TEXTLIST S3_Alarms
  0 = 'Station 3 Clamp A1 Failed to Advance... Check Q1.0...' | German: 'S3 0 Row 1 Failed To Advance.. Check Qxxx.x German' | French: 'S3 0 Row 1 Failed To Advance.. Check Qxxx.x French' | 汉语: '汉语'
  1 = 'Station 3 Clamp A1 Failed to Return... Check Q1.1...' | German: 'S3 1 Row 1 Failed To Return.. Check Qxxx.x German' | French: 'S3 1 Row 1 Failed To Return.. Check Qxxx.x French' | 汉语: '汉语'
  2 = 'Station 3 Clamp A1 Lost Advanced... Check I1.0...' | German: 'S3 2 Row 1 Lost Advance Position... Check Ixxx.x German' | French: 'S3 2 Row 1 Lost Advance Position... Check Ixxx.x French' | 汉语: '汉语'
  3 = 'Station 3 Clamp A1 Lost Returned... Check I1.1...' | German: 'S3 3 Row 1 Lost Return Position... Check Ixxx.x German' | French: 'S3 3 Row 1 Lost Return Position... Check Ixxx.x French' | 汉语: '汉语'
  4 = 'Station 3 Clamp A1 Switch Fault... Check I1.0, I1.1...' | German: 'S3 4 Row 1 Switch Fault... Check Ixxx.x / Ixxx.x German' | French: 'S3 4 Row 1 Switch Fault... Check Ixxx.x / Ixxx.x French' | 汉语: '汉语'
  5 = 'Spare' | German: 'S3 5 Row 1 Spare Message German' | French: 'S3 5 Row 1 Spare Message French'
  6 = 'Spare' | German: 'S3 6 Row 1 Spare Message German' | French: 'S3 6 Row 1 Spare Message French'
  7 = 'Spare' | German: 'S3 7 Row 1 Spare Message German' | French: 'S3 7 Row 1 Spare Message French'
  8 = 'Spare' | German: 'S3 8 Row 1 Spare Message German' | French: 'S3 8 Row 1 Spare Message French'
  9 = 'Spare' | German: 'S3 9 Row 1 Spare Message German' | French: 'S3 9 Row 1 Spare Message French'
  10 = 'Lock Cylinder A2 Failed to Lock... Check Q1.2...' | German: 'S3 10 Row 2 Failed To Advance.. Check Qxxx.x German' | French: 'S3 10 Row 2 Failed To Advance.. Check Qxxx.x French'
  11 = 'Lock Cylinder A2 Failed to Unlock... Check Q1.3...' | German: 'S3 11 Row 2 Failed To Return.. Check Qxxx.x German' | French: 'S3 11 Row 2 Failed To Return.. Check Qxxx.x French'
  12 = 'Lock Cylinder A2 Lost Locked... Check I1.2...' | German: 'S3 12 Row 2 Lost Advance Position... Check Ixxx.x German' | French: 'S3 12 Row 2 Lost Advance Position... Check Ixxx.x French'
  13 = 'Lock Cylinder A2 Lost Unlocked... Check I1.3...' | German: 'S3 13 Row 2 Lost Return Position... Check Ixxx.x German' | French: 'S3 13 Row 2 Lost Return Position... Check Ixxx.x French'
  14 = 'Lock Cylinder A2 Switch Fault... Check I1.2, I1.3...' | German: 'S3 14 Row 2 Switch Fault... Check Ixxx.x / Ixxx.x German' | French: 'S3 14 Row 2 Switch Fault... Check Ixxx.x / Ixxx.x French'
  15 = 'Spare' | German: 'S3 15 Row 2 Spare Message German' | French: 'S3 15 Row 2 Spare Message French'
  16 = 'Spare' | German: 'S3 16 Row 2 Spare Message German' | French: 'S3 16 Row 2 Spare Message French'
  17 = 'Spare' | German: 'S3 17 Row 2 Spare Message German' | French: 'S3 17 Row 2 Spare Message French'
  18 = 'Spare' | German: 'S3 18 Row 2 Spare Message German' | French: 'S3 18 Row 2 Spare Message French'
  19 = 'Spare' | German: 'S3 19 Row 2 Spare Message German' | French: 'S3 19 Row 2 Spare Message French'
  20 = 'Urger Cylinder A3 Failed to Urge... Check Q1.4...' | German: 'S3 20 Row 3 Failed To Advance.. Check Qxxx.x German' | French: 'S3 20 Row 3 Failed To Advance.. Check Qxxx.x French'
  21 = 'Urger Cylinder A3 Failed to Return... Check Q1.5...' | German: 'S3 21 Row 3 Failed To Return.. Check Qxxx.x German' | French: 'S3 21 Row 3 Failed To Return.. Check Qxxx.x French'
  22 = 'Urger Cylinder A3 Lost Urged... Check I1.4...' | German: 'S3 22 Row 3 Lost Advance Position... Check Ixxx.x German' | French: 'S3 22 Row 3 Lost Advance Position... Check Ixxx.x French'
  23 = 'Urger Cylinder A3 Lost Returned... Check I1.5...' | German: 'S3 23 Row 3 Lost Return Position... Check Ixxx.x German' | French: 'S3 23 Row 3 Lost Return Position... Check Ixxx.x French'
  24 = 'Urger Cylinder A3 Switch Fault... Check I1.4, I1.5...' | German: 'S3 24 Row 3 Switch Fault... Check Ixxx.x / Ixxx.x German' | French: 'S3 24 Row 3 Switch Fault... Check Ixxx.x / Ixxx.x French'
  25 = 'Spare' | German: 'S3 25 Row 3 Spare Message German' | French: 'S3 25 Row 3 Spare Message French'
  26 = 'Spare' | German: 'S3 26 Row 3 Spare Message German' | French: 'S3 26 Row 3 Spare Message French'
  27 = 'Spare' | German: 'S3 27 Row 3 Spare Message German' | French: 'S3 27 Row 3 Spare Message French'
  28 = 'Spare' | German: 'S3 28 Row 3 Spare Message German' | French: 'S3 28 Row 3 Spare Message French'
  29 = 'Spare' | German: 'S3 29 Row 3 Spare Message German' | French: 'S3 29 Row 3 Spare Message French'
  30 = 'Clamp Cylinder A1 Failed to Advance... Check Q1.0...' | German: 'S3 30 Row 4 Failed To Advance.. Check Qxxx.x German' | French: 'S3 30 Row 4 Failed To Advance.. Check Qxxx.x French'
  31 = 'Clamp Cylinder A1 Failed to Return... Check Q1.1...' | German: 'S3 31 Row 4 Failed To Return.. Check Qxxx.x German' | French: 'S3 31 Row 4 Failed To Return.. Check Qxxx.x French'
  32 = 'Clamp Cylinder A1 Lost Advanced... Check I1.0...' | German: 'S3 32 Row 4 Lost Advance Position... Check Ixxx.x German' | French: 'S3 32 Row 4 Lost Advance Position... Check Ixxx.x French'
  33 = 'Clamp Cylinder A1 Lost Returned... Check I1.1...' | German: 'S3 33 Row 4 Lost Return Position... Check Ixxx.x German' | French: 'S3 33 Row 4 Lost Return Position... Check Ixxx.x French'
  34 = 'Clamp Cylinder A1 Switch Fault... Check I1.0, I1.1...' | German: 'S3 34 Row 4 Switch Fault... Check Ixxx.x / Ixxx.x German' | French: 'S3 34 Row 4 Switch Fault... Check Ixxx.x / Ixxx.x French'
  35 = 'Spare' | German: 'S3 35 Row 4 Spare Message German' | French: 'S3 35 Row 4 Spare Message French'
  36 = 'Spare' | German: 'S3 36 Row 4 Spare Message German' | French: 'S3 36 Row 4 Spare Message French'
  37 = 'Spare' | German: 'S3 37 Row 4 Spare Message German' | French: 'S3 37 Row 4 Spare Message French'
  38 = 'Spare' | German: 'S3 38 Row 4 Spare Message German' | French: 'S3 38 Row 4 Spare Message French'
  39 = 'Spare' | German: 'S3 39 Row 4 Spare Message German' | French: 'S3 39 Row 4 Spare Message French'
  40 = 'Clamp Cylinder A1 Failed to Advance... Check Q1.0...' | German: 'S3 40 Row 5 Failed To Advance.. Check Qxxx.x German' | French: 'S3 40 Row 5 Failed To Advance.. Check Qxxx.x French'
  41 = 'Clamp Cylinder A1 Failed to Return... Check Q1.1...' | German: 'S3 41 Row 5 Failed To Return.. Check Qxxx.x German' | French: 'S3 41 Row 5 Failed To Return.. Check Qxxx.x French'
  42 = 'Clamp Cylinder A1 Lost Advanced... Check I1.0...' | German: 'S3 42 Row 5 Lost Advance Position... Check Ixxx.x German' | French: 'S3 42 Row 5 Lost Advance Position... Check Ixxx.x French'
  43 = 'Clamp Cylinder A1 Lost Returned... Check I1.1...' | German: 'S3 43 Row 5 Lost Return Position... Check Ixxx.x German' | French: 'S3 43 Row 5 Lost Return Position... Check Ixxx.x French'
  44 = 'Clamp Cylinder A1 Switch Fault... Check I1.0, I1.1...' | German: 'S3 44 Row 5 Switch Fault... Check Ixxx.x / Ixxx.x German' | French: 'S3 44 Row 5 Switch Fault... Check Ixxx.x / Ixxx.x French'
  45 = 'Spare' | German: 'S3 45 Row 5 Spare Message German' | French: 'S3 45 Row 5 Spare Message French'
  46 = 'Spare' | German: 'S3 46 Row 5 Spare Message German' | French: 'S3 46 Row 5 Spare Message French'
  47 = 'Spare' | German: 'S3 47 Row 5 Spare Message German' | French: 'S3 47 Row 5 Spare Message French'
  48 = 'Spare' | German: 'S3 48 Row 5 Spare Message German' | French: 'S3 48 Row 5 Spare Message French'
  49 = 'Spare' | German: 'S3 49 Row 5 Spare Message German' | French: 'S3 49 Row 5 Spare Message French'
  50 = 'Clamp Cylinder A1 Failed to Advance... Check Q1.0...' | German: 'S3 50 Row 6 Failed To Advance.. Check Qxxx.x German' | French: 'S3 50 Row 6 Failed To Advance.. Check Qxxx.x French'
  51 = 'Clamp Cylinder A1 Failed to Return... Check Q1.1...' | German: 'S3 51 Row 6 Failed To Return.. Check Qxxx.x German' | French: 'S3 51 Row 6 Failed To Return.. Check Qxxx.x French'
  52 = 'Clamp Cylinder A1 Lost Advanced... Check I1.0...' | German: 'S3 52 Row 6 Lost Advance Position... Check Ixxx.x German' | French: 'S3 52 Row 6 Lost Advance Position... Check Ixxx.x French'
  53 = 'Clamp Cylinder A1 Lost Returned... Check I1.1...' | German: 'S3 53 Row 6 Lost Return Position... Check Ixxx.x German' | French: 'S3 53 Row 6 Lost Return Position... Check Ixxx.x French'
  54 = 'Clamp Cylinder A1 Switch Fault... Check I1.0, I1.1...' | German: 'S3 54 Row 6 Switch Fault... Check Ixxx.x / Ixxx.x German' | French: 'S3 54 Row 6 Switch Fault... Check Ixxx.x / Ixxx.x French'
  55 = 'Spare' | German: 'S3 55 Row 6 Spare Message German' | French: 'S3 55 Row 6 Spare Message French'
  56 = 'Spare' | German: 'S3 56 Row 6 Spare Message German' | French: 'S3 56 Row 6 Spare Message French'
  57 = 'Spare' | German: 'S3 57 Row 6 Spare Message German' | French: 'S3 57 Row 6 Spare Message French'
  58 = 'Spare' | German: 'S3 58 Row 6 Spare Message German' | French: 'S3 58 Row 6 Spare Message French'
  59 = 'Spare' | German: 'S3 59 Row 6 Spare Message German' | French: 'S3 59 Row 6 Spare Message French'
  60 = 'Clamp Cylinder A1 Failed to Advance... Check Q1.0...' | German: 'S3 60 Row 7 Failed To Advance.. Check Qxxx.x German' | French: 'S3 60 Row 7 Failed To Advance.. Check Qxxx.x French'
  61 = 'Clamp Cylinder A1 Failed to Return... Check Q1.1...' | German: 'S3 61 Row 7 Failed To Return.. Check Qxxx.x German' | French: 'S3 61 Row 7 Failed To Return.. Check Qxxx.x French'
  62 = 'Clamp Cylinder A1 Lost Advanced... Check I1.0...' | German: 'S3 62 Row 7 Lost Advance Position... Check Ixxx.x German' | French: 'S3 62 Row 7 Lost Advance Position... Check Ixxx.x French'
  63 = 'Clamp Cylinder A1 Lost Returned... Check I1.1...' | German: 'S3 63 Row 7 Lost Return Position... Check Ixxx.x German' | French: 'S3 63 Row 7 Lost Return Position... Check Ixxx.x French'
  64 = 'Clamp Cylinder A1 Switch Fault... Check I1.0, I1.1...' | German: 'S3 64 Row 7 Switch Fault... Check Ixxx.x / Ixxx.x German' | French: 'S3 64 Row 7 Switch Fault... Check Ixxx.x / Ixxx.x French'
  65 = 'Spare' | German: 'S3 65 Row 7 Spare Message German' | French: 'S3 65 Row 7 Spare Message French'
  66 = 'Spare' | German: 'S3 66 Row 7 Spare Message German' | French: 'S3 66 Row 7 Spare Message French'
  67 = 'Spare' | German: 'S3 67 Row 7 Spare Message German' | French: 'S3 67 Row 7 Spare Message French'
  68 = 'Spare' | German: 'S3 68 Row 7 Spare Message German' | French: 'S3 68 Row 7 Spare Message French'
  69 = 'Spare' | German: 'S3 69 Row 7 Spare Message German' | French: 'S3 69 Row 7 Spare Message French'
  70 = 'Clamp Cylinder A1 Failed to Advance... Check Q1.0...' | German: 'S3 70 Row 8 Failed To Advance.. Check Qxxx.x German' | French: 'S3 70 Row 8 Failed To Advance.. Check Qxxx.x French'
  71 = 'Clamp Cylinder A1 Failed to Return... Check Q1.1...' | German: 'S3 71 Row 8 Failed To Return.. Check Qxxx.x German' | French: 'S3 71 Row 8 Failed To Return.. Check Qxxx.x French'
  72 = 'Clamp Cylinder A1 Lost Advanced... Check I1.0...' | German: 'S3 72 Row 8 Lost Advance Position... Check Ixxx.x German' | French: 'S3 72 Row 8 Lost Advance Position... Check Ixxx.x French'
  73 = 'Clamp Cylinder A1 Lost Returned... Check I1.1...' | German: 'S3 73 Row 8 Lost Return Position... Check Ixxx.x German' | French: 'S3 73 Row 8 Lost Return Position... Check Ixxx.x French'
  74 = 'Clamp Cylinder A1 Switch Fault... Check I1.0, I1.1...' | German: 'S3 74 Row 8 Switch Fault... Check Ixxx.x / Ixxx.x German' | French: 'S3 74 Row 8 Switch Fault... Check Ixxx.x / Ixxx.x French'
  75 = 'Spare' | German: 'S3 75 Row 8 Spare Message German' | French: 'S3 75 Row 8 Spare Message French'
  76 = 'Spare' | German: 'S3 76 Row 8 Spare Message German' | French: 'S3 76 Row 8 Spare Message French'
  77 = 'Spare' | German: 'S3 77 Row 8 Spare Message German' | French: 'S3 77 Row 8 Spare Message French'
  78 = 'Spare' | German: 'S3 78 Row 8 Spare Message German' | French: 'S3 78 Row 8 Spare Message French'
  79 = 'Spare' | German: 'S3 79 Row 8 Spare Message German' | French: 'S3 79 Row 8 Spare Message French'
  80 = 'Clamp Cylinder A1 Failed to Advance... Check Q1.0...' | German: 'S3 80 Row 9 Failed To Advance.. Check Qxxx.x German' | French: 'S3 80 Row 9 Failed To Advance.. Check Qxxx.x French'
  81 = 'Clamp Cylinder A1 Failed to Return... Check Q1.1...' | German: 'S3 81 Row 9 Failed To Return.. Check Qxxx.x German' | French: 'S3 81 Row 9 Failed To Return.. Check Qxxx.x French'
  82 = 'Clamp Cylinder A1 Lost Advanced... Check I1.0...' | German: 'S3 82 Row 9 Lost Advance Position... Check Ixxx.x German' | French: 'S3 82 Row 9 Lost Advance Position... Check Ixxx.x French'
  83 = 'Clamp Cylinder A1 Lost Returned... Check I1.1...' | German: 'S3 83 Row 9 Lost Return Position... Check Ixxx.x German' | French: 'S3 83 Row 9 Lost Return Position... Check Ixxx.x French'
  84 = 'Clamp Cylinder A1 Switch Fault... Check I1.0, I1.1...' | German: 'S3 84 Row 9 Switch Fault... Check Ixxx.x / Ixxx.x German' | French: 'S3 84 Row 9 Switch Fault... Check Ixxx.x / Ixxx.x French'
  85 = 'Spare' | German: 'S3 85 Row 9 Spare Message German' | French: 'S3 85 Row 9 Spare Message French'
  86 = 'Spare' | German: 'S3 86 Row 9 Spare Message German' | French: 'S3 86 Row 9 Spare Message French'
  87 = 'Spare' | German: 'S3 87 Row 9 Spare Message German' | French: 'S3 87 Row 9 Spare Message French'
  88 = 'Spare' | German: 'S3 88 Row 9 Spare Message German' | French: 'S3 88 Row 9 Spare Message French'
  89 = 'Spare' | German: 'S3 89 Row 9 Spare Message German' | French: 'S3 89 Row 9 Spare Message French'
  90 = 'Clamp Cylinder A1 Failed to Advance... Check Q1.0...' | German: 'S3 90 Row 10 Failed To Advance.. Check Qxxx.x German' | French: 'S3 90 Row 10 Failed To Advance.. Check Qxxx.x French'
  91 = 'Clamp Cylinder A1 Failed to Return... Check Q1.1...' | German: 'S3 91 Row 10 Failed To Return.. Check Qxxx.x German' | French: 'S3 91 Row 10 Failed To Return.. Check Qxxx.x French'
  92 = 'Clamp Cylinder A1 Lost Advanced... Check I1.0...' | German: 'S3 92 Row 10 Lost Advance Position... Check Ixxx.x German' | French: 'S3 92 Row 10 Lost Advance Position... Check Ixxx.x French'
  93 = 'Clamp Cylinder A1 Lost Returned... Check I1.1...' | German: 'S3 93 Row 10 Lost Return Position... Check Ixxx.x German' | French: 'S3 93 Row 10 Lost Return Position... Check Ixxx.x French'
  94 = 'Clamp Cylinder A1 Switch Fault... Check I1.0, I1.1...' | German: 'S3 94 Row 10 Switch Fault... Check Ixxx.x / Ixxx.x German' | French: 'S3 94 Row 10 Switch Fault... Check Ixxx.x / Ixxx.x French'
  95 = 'Spare' | German: 'S3 95 Row 10 Spare Message German' | French: 'S3 95 Row 10 Spare Message French'
  96 = 'Spare' | German: 'S3 96 Row 10 Spare Message German' | French: 'S3 96 Row 10 Spare Message French'
  97 = 'Spare' | German: 'S3 97 Row 10 Spare Message German' | French: 'S3 97 Row 10 Spare Message French'
  98 = 'Spare' | German: 'S3 98 Row 10 Spare Message German' | French: 'S3 98 Row 10 Spare Message French'
  99 = 'Spare' | German: 'S3 99 Row 10 Spare Message German' | French: 'S3 99 Row 10 Spare Message French'
  100 = 'Clamp Cylinder A1 Failed to Advance... Check Q1.0...' | German: 'S3 100 Row 11 Failed To Advance.. Check Qxxx.x German' | French: 'S3 100 Row 11 Failed To Advance.. Check Qxxx.x French'
  101 = 'Clamp Cylinder A1 Failed to Return... Check Q1.1...' | German: 'S3 101 Row 11 Failed To Return.. Check Qxxx.x German' | French: 'S3 101 Row 11 Failed To Return.. Check Qxxx.x French'
  102 = 'Clamp Cylinder A1 Lost Advanced... Check I1.0...' | German: 'S3 102 Row 11 Lost Advance Position... Check Ixxx.x German' | French: 'S3 102 Row 11 Lost Advance Position... Check Ixxx.x French'
  103 = 'Clamp Cylinder A1 Lost Returned... Check I1.1...' | German: 'S3 103 Row 11 Lost Return Position... Check Ixxx.x German' | French: 'S3 103 Row 11 Lost Return Position... Check Ixxx.x French'
  104 = 'Clamp Cylinder A1 Switch Fault... Check I1.0, I1.1...' | German: 'S3 104 Row 11 Switch Fault... Check Ixxx.x / Ixxx.x German' | French: 'S3 104 Row 11 Switch Fault... Check Ixxx.x / Ixxx.x French'
  105 = 'Spare' | German: 'S3 105 Row 11 Spare Message German' | French: 'S3 105 Row 11 Spare Message French'
  106 = 'Spare' | German: 'S3 106 Row 11 Spare Message German' | French: 'S3 106 Row 11 Spare Message French'
  107 = 'Spare' | German: 'S3 107 Row 11 Spare Message German' | French: 'S3 107 Row 11 Spare Message French'
  108 = 'Spare' | German: 'S3 108 Row 11 Spare Message German' | French: 'S3 108 Row 11 Spare Message French'
  109 = 'Spare' | German: 'S3 109 Row 11 Spare Message German' | French: 'S3 109 Row 11 Spare Message French'
  110 = 'Clamp Cylinder A1 Failed to Advance... Check Q1.0...' | German: 'S3 110 Row 12 Failed To Advance.. Check Qxxx.x German' | French: 'S3 110 Row 12 Failed To Advance.. Check Qxxx.x French'
  111 = 'Clamp Cylinder A1 Failed to Return... Check Q1.1...' | German: 'S3 111 Row 12 Failed To Return.. Check Qxxx.x German' | French: 'S3 111 Row 12 Failed To Return.. Check Qxxx.x French'
  112 = 'Clamp Cylinder A1 Lost Advanced... Check I1.0...' | German: 'S3 112 Row 12 Lost Advance Position... Check Ixxx.x German' | French: 'S3 112 Row 12 Lost Advance Position... Check Ixxx.x French'
  113 = 'Clamp Cylinder A1 Lost Returned... Check I1.1...' | German: 'S3 113 Row 12 Lost Return Position... Check Ixxx.x German' | French: 'S3 113 Row 12 Lost Return Position... Check Ixxx.x French'
  114 = 'Clamp Cylinder A1 Switch Fault... Check I1.0, I1.1...' | German: 'S3 114 Row 12 Switch Fault... Check Ixxx.x / Ixxx.x German' | French: 'S3 114 Row 12 Switch Fault... Check Ixxx.x / Ixxx.x French'
  115 = 'Spare' | German: 'S3 115 Row 12 Spare Message German' | French: 'S3 115 Row 12 Spare Message French'
  116 = 'Spare' | German: 'S3 116 Row 12 Spare Message German' | French: 'S3 116 Row 12 Spare Message French'
  117 = 'Spare' | German: 'S3 117 Row 12 Spare Message German' | French: 'S3 117 Row 12 Spare Message French'
  118 = 'Spare' | German: 'S3 118 Row 12 Spare Message German' | French: 'S3 118 Row 12 Spare Message French'
  119 = 'Spare' | German: 'S3 119 Row 12 Spare Message German' | French: 'S3 119 Row 12 Spare Message French'
  120 = 'Clamp Cylinder A1 Failed to Advance... Check Q1.0...' | German: 'S3 120 Row 13 Failed To Advance.. Check Qxxx.x German' | French: 'S3 120 Row 13 Failed To Advance.. Check Qxxx.x French'
  121 = 'Clamp Cylinder A1 Failed to Return... Check Q1.1...' | German: 'S3 121 Row 13 Failed To Return.. Check Qxxx.x German' | French: 'S3 121 Row 13 Failed To Return.. Check Qxxx.x French'
  122 = 'Clamp Cylinder A1 Lost Advanced... Check I1.0...' | German: 'S3 122 Row 13 Lost Advance Position... Check Ixxx.x German' | French: 'S3 122 Row 13 Lost Advance Position... Check Ixxx.x French'
  123 = 'Clamp Cylinder A1 Lost Returned... Check I1.1...' | German: 'S3 123 Row 13 Lost Return Position... Check Ixxx.x German' | French: 'S3 123 Row 13 Lost Return Position... Check Ixxx.x French'
  124 = 'Clamp Cylinder A1 Switch Fault... Check I1.0, I1.1...' | German: 'S3 124 Row 13 Switch Fault... Check Ixxx.x / Ixxx.x German' | French: 'S3 124 Row 13 Switch Fault... Check Ixxx.x / Ixxx.x French'
  125 = 'Spare' | German: 'S3 125 Row 13 Spare Message German' | French: 'S3 125 Row 13 Spare Message French'
  126 = 'Spare' | German: 'S3 126 Row 13 Spare Message German' | French: 'S3 126 Row 13 Spare Message French'
  127 = 'Spare' | German: 'S3 127 Row 13 Spare Message German' | French: 'S3 127 Row 13 Spare Message French'
  128 = 'Spare' | German: 'S3 128 Row 13 Spare Message German' | French: 'S3 128 Row 13 Spare Message French'
  129 = 'Spare' | German: 'S3 129 Row 13 Spare Message German' | French: 'S3 129 Row 13 Spare Message French'
  130 = 'Clamp Cylinder A1 Failed to Advance... Check Q1.0...' | German: 'S3 130 Row 14 Failed To Advance.. Check Qxxx.x German' | French: 'S3 130 Row 14 Failed To Advance.. Check Qxxx.x French'
  131 = 'Clamp Cylinder A1 Failed to Return... Check Q1.1...' | German: 'S3 131 Row 14 Failed To Return.. Check Qxxx.x German' | French: 'S3 131 Row 14 Failed To Return.. Check Qxxx.x French'
  132 = 'Clamp Cylinder A1 Lost Advanced... Check I1.0...' | German: 'S3 132 Row 14 Lost Advance Position... Check Ixxx.x German' | French: 'S3 132 Row 14 Lost Advance Position... Check Ixxx.x French'
  133 = 'Clamp Cylinder A1 Lost Returned... Check I1.1...' | German: 'S3 133 Row 14 Lost Return Position... Check Ixxx.x German' | French: 'S3 133 Row 14 Lost Return Position... Check Ixxx.x French'
  134 = 'Clamp Cylinder A1 Switch Fault... Check I1.0, I1.1...' | German: 'S3 134 Row 14 Switch Fault... Check Ixxx.x / Ixxx.x German' | French: 'S3 134 Row 14 Switch Fault... Check Ixxx.x / Ixxx.x French'
  135 = 'Spare' | German: 'S3 135 Row 14 Spare Message German' | French: 'S3 135 Row 14 Spare Message French'
  136 = 'Spare' | German: 'S3 136 Row 14 Spare Message German' | French: 'S3 136 Row 14 Spare Message French'
  137 = 'Spare' | German: 'S3 137 Row 14 Spare Message German' | French: 'S3 137 Row 14 Spare Message French'
  138 = 'Spare' | German: 'S3 138 Row 14 Spare Message German' | French: 'S3 138 Row 14 Spare Message French'
  139 = 'Spare' | German: 'S3 139 Row 14 Spare Message German' | French: 'S3 139 Row 14 Spare Message French'
  140 = 'Clamp Cylinder A1 Failed to Advance... Check Q1.0...' | German: 'S3 140 Row 15 Failed To Advance.. Check Qxxx.x German' | French: 'S3 140 Row 15 Failed To Advance.. Check Qxxx.x French'
  141 = 'Clamp Cylinder A1 Failed to Return... Check Q1.1...' | German: 'S3 141 Row 15 Failed To Return.. Check Qxxx.x German' | French: 'S3 141 Row 15 Failed To Return.. Check Qxxx.x French'
  142 = 'Clamp Cylinder A1 Lost Advanced... Check I1.0...' | German: 'S3 142 Row 15 Lost Advance Position... Check Ixxx.x German' | French: 'S3 142 Row 15 Lost Advance Position... Check Ixxx.x French'
  143 = 'Clamp Cylinder A1 Lost Returned... Check I1.1...' | German: 'S3 143 Row 15 Lost Return Position... Check Ixxx.x German' | French: 'S3 143 Row 15 Lost Return Position... Check Ixxx.x French'
  144 = 'Clamp Cylinder A1 Switch Fault... Check I1.0, I1.1...' | German: 'S3 144 Row 15 Switch Fault... Check Ixxx.x / Ixxx.x German' | French: 'S3 144 Row 15 Switch Fault... Check Ixxx.x / Ixxx.x French'
  145 = 'Spare' | German: 'S3 145 Row 15 Spare Message German' | French: 'S3 145 Row 15 Spare Message French'
  146 = 'Spare' | German: 'S3 146 Row 15 Spare Message German' | French: 'S3 146 Row 15 Spare Message French'
  147 = 'Spare' | German: 'S3 147 Row 15 Spare Message German' | French: 'S3 147 Row 15 Spare Message French'
  148 = 'Spare' | German: 'S3 148 Row 15 Spare Message German' | French: 'S3 148 Row 15 Spare Message French'
  149 = 'Spare' | German: 'S3 149 Row 15 Spare Message German' | French: 'S3 149 Row 15 Spare Message French'
  150 = 'Clamp Cylinder A1 Failed to Advance... Check Q1.0...' | German: 'S3 150 Row 16 Failed To Advance.. Check Qxxx.x German' | French: 'S3 150 Row 16 Failed To Advance.. Check Qxxx.x French'
  151 = 'Clamp Cylinder A1 Failed to Return... Check Q1.1...' | German: 'S3 151 Row 16 Failed To Return.. Check Qxxx.x German' | French: 'S3 151 Row 16 Failed To Return.. Check Qxxx.x French'
  152 = 'Clamp Cylinder A1 Lost Advanced... Check I1.0...' | German: 'S3 152 Row 16 Lost Advance Position... Check Ixxx.x German' | French: 'S3 152 Row 16 Lost Advance Position... Check Ixxx.x French'
  153 = 'Clamp Cylinder A1 Lost Returned... Check I1.1...' | German: 'S3 153 Row 16 Lost Return Position... Check Ixxx.x German' | French: 'S3 153 Row 16 Lost Return Position... Check Ixxx.x French'
  154 = 'Clamp Cylinder A1 Switch Fault... Check I1.0, I1.1...' | German: 'S3 154 Row 16 Switch Fault... Check Ixxx.x / Ixxx.x German' | French: 'S3 154 Row 16 Switch Fault... Check Ixxx.x / Ixxx.x French'
  155 = 'Spare' | German: 'S3 155 Row 16 Spare Message German' | French: 'S3 155 Row 16 Spare Message French'
  156 = 'Spare' | German: 'S3 156 Row 16 Spare Message German' | French: 'S3 156 Row 16 Spare Message French'
  157 = 'Spare' | German: 'S3 157 Row 16 Spare Message German' | French: 'S3 157 Row 16 Spare Message French'
  158 = 'Spare' | German: 'S3 158 Row 16 Spare Message German' | French: 'S3 158 Row 16 Spare Message French'
  159 = 'Spare' | German: 'S3 159 Row 16 Spare Message German' | French: 'S3 159 Row 16 Spare Message French'
  160 = 'Clamp Cylinder A1 Failed to Advance... Check Q1.0...' | German: 'S3 160 Row 17 Failed To Advance.. Check Qxxx.x German' | French: 'S3 160 Row 17 Failed To Advance.. Check Qxxx.x French'
  161 = 'Clamp Cylinder A1 Failed to Return... Check Q1.1...' | German: 'S3 161 Row 17 Failed To Return.. Check Qxxx.x German' | French: 'S3 161 Row 17 Failed To Return.. Check Qxxx.x French'
  162 = 'Clamp Cylinder A1 Lost Advanced... Check I1.0...' | German: 'S3 162 Row 17 Lost Advance Position... Check Ixxx.x German' | French: 'S3 162 Row 17 Lost Advance Position... Check Ixxx.x French'
  163 = 'Clamp Cylinder A1 Lost Returned... Check I1.1...' | German: 'S3 163 Row 17 Lost Return Position... Check Ixxx.x German' | French: 'S3 163 Row 17 Lost Return Position... Check Ixxx.x French'
  164 = 'Clamp Cylinder A1 Switch Fault... Check I1.0, I1.1...' | German: 'S3 164 Row 17 Switch Fault... Check Ixxx.x / Ixxx.x German' | French: 'S3 164 Row 17 Switch Fault... Check Ixxx.x / Ixxx.x French'
  165 = 'Spare' | German: 'S3 165 Row 17 Spare Message German' | French: 'S3 165 Row 17 Spare Message French'
  166 = 'Spare' | German: 'S3 166 Row 17 Spare Message German' | French: 'S3 166 Row 17 Spare Message French'
  167 = 'Spare' | German: 'S3 167 Row 17 Spare Message German' | French: 'S3 167 Row 17 Spare Message French'
  168 = 'Spare' | German: 'S3 168 Row 17 Spare Message German' | French: 'S3 168 Row 17 Spare Message French'
  169 = 'Spare' | German: 'S3 169 Row 17 Spare Message German' | French: 'S3 169 Row 17 Spare Message French'
  170 = 'Clamp Cylinder A1 Failed to Advance... Check Q1.0...' | German: 'S3 170 Row 18 Failed To Advance.. Check Qxxx.x German' | French: 'S3 170 Row 18 Failed To Advance.. Check Qxxx.x French'
  171 = 'Clamp Cylinder A1 Failed to Return... Check Q1.1...' | German: 'S3 171 Row 18 Failed To Return.. Check Qxxx.x German' | French: 'S3 171 Row 18 Failed To Return.. Check Qxxx.x French'
  172 = 'Clamp Cylinder A1 Lost Advanced... Check I1.0...' | German: 'S3 172 Row 18 Lost Advance Position... Check Ixxx.x German' | French: 'S3 172 Row 18 Lost Advance Position... Check Ixxx.x French'
  173 = 'Clamp Cylinder A1 Lost Returned... Check I1.1...' | German: 'S3 173 Row 18 Lost Return Position... Check Ixxx.x German' | French: 'S3 173 Row 18 Lost Return Position... Check Ixxx.x French'
  174 = 'Clamp Cylinder A1 Switch Fault... Check I1.0, I1.1...' | German: 'S3 174 Row 18 Switch Fault... Check Ixxx.x / Ixxx.x German' | French: 'S3 174 Row 18 Switch Fault... Check Ixxx.x / Ixxx.x French'
  175 = 'Spare' | German: 'S3 175 Row 18 Spare Message German' | French: 'S3 175 Row 18 Spare Message French'
  176 = 'Spare' | German: 'S3 176 Row 18 Spare Message German' | French: 'S3 176 Row 18 Spare Message French'
  177 = 'Spare' | German: 'S3 177 Row 18 Spare Message German' | French: 'S3 177 Row 18 Spare Message French'
  178 = 'Spare' | German: 'S3 178 Row 18 Spare Message German' | French: 'S3 178 Row 18 Spare Message French'
  179 = 'Spare' | German: 'S3 179 Row 18 Spare Message German' | French: 'S3 179 Row 18 Spare Message French'
  180 = 'Clamp Cylinder A1 Failed to Advance... Check Q1.0...' | German: 'S3 180 Row 19 Failed To Advance.. Check Qxxx.x German' | French: 'S3 180 Row 19 Failed To Advance.. Check Qxxx.x French'
  181 = 'Clamp Cylinder A1 Failed to Return... Check Q1.1...' | German: 'S3 181 Row 19 Failed To Return.. Check Qxxx.x German' | French: 'S3 181 Row 19 Failed To Return.. Check Qxxx.x French'
  182 = 'Clamp Cylinder A1 Lost Advanced... Check I1.0...' | German: 'S3 182 Row 19 Lost Advance Position... Check Ixxx.x German' | French: 'S3 182 Row 19 Lost Advance Position... Check Ixxx.x French'
  183 = 'Clamp Cylinder A1 Lost Returned... Check I1.1...' | German: 'S3 183 Row 19 Lost Return Position... Check Ixxx.x German' | French: 'S3 183 Row 19 Lost Return Position... Check Ixxx.x French'
  184 = 'Clamp Cylinder A1 Switch Fault... Check I1.0, I1.1...' | German: 'S3 184 Row 19 Switch Fault... Check Ixxx.x / Ixxx.x German' | French: 'S3 184 Row 19 Switch Fault... Check Ixxx.x / Ixxx.x French'
  185 = 'Spare' | German: 'S3 185 Row 19 Spare Message German' | French: 'S3 185 Row 19 Spare Message French'
  186 = 'Spare' | German: 'S3 186 Row 19 Spare Message German' | French: 'S3 186 Row 19 Spare Message French'
  187 = 'Spare' | German: 'S3 187 Row 19 Spare Message German' | French: 'S3 187 Row 19 Spare Message French'
  188 = 'Spare' | German: 'S3 188 Row 19 Spare Message German' | French: 'S3 188 Row 19 Spare Message French'
  189 = 'Spare' | German: 'S3 189 Row 19 Spare Message German' | French: 'S3 189 Row 19 Spare Message French'
  190 = 'Clamp Cylinder A1 Failed to Advance... Check Q1.0...' | German: 'S3 190 Row 20 Failed To Advance.. Check Qxxx.x German' | French: 'S3 190 Row 20 Failed To Advance.. Check Qxxx.x French'
  191 = 'Clamp Cylinder A1 Failed to Return... Check Q1.1...' | German: 'S3 191 Row 20 Failed To Return.. Check Qxxx.x German' | French: 'S3 191 Row 20 Failed To Return.. Check Qxxx.x French'
  192 = 'Clamp Cylinder A1 Lost Advanced... Check I1.0...' | German: 'S3 192 Row 20 Lost Advance Position... Check Ixxx.x German' | French: 'S3 192 Row 20 Lost Advance Position... Check Ixxx.x French'
  193 = 'Clamp Cylinder A1 Lost Returned... Check I1.1...' | German: 'S3 193 Row 20 Lost Return Position... Check Ixxx.x German' | French: 'S3 193 Row 20 Lost Return Position... Check Ixxx.x French'
  194 = 'Clamp Cylinder A1 Switch Fault... Check I1.0, I1.1...' | German: 'S3 194 Row 20 Switch Fault... Check Ixxx.x / Ixxx.x German' | French: 'S3 194 Row 20 Switch Fault... Check Ixxx.x / Ixxx.x French'
  195 = 'Spare' | German: 'S3 195 Row 20 Spare Message German' | French: 'S3 195 Row 20 Spare Message French'
  196 = 'Spare' | German: 'S3 196 Row 20 Spare Message German' | French: 'S3 196 Row 20 Spare Message French'
  197 = 'Spare' | German: 'S3 197 Row 20 Spare Message German' | French: 'S3 197 Row 20 Spare Message French'
  198 = 'Spare' | German: 'S3 198 Row 20 Spare Message German' | French: 'S3 198 Row 20 Spare Message French'
  199 = 'Spare' | German: 'S3 199 Row 20 Spare Message German' | French: 'S3 199 Row 20 Spare Message French'
  200 = 'Clamp Cylinder A1 Failed to Advance... Check Q1.0...' | German: 'S3 200 Row 21 Failed To Advance.. Check Qxxx.x German' | French: 'S3 200 Row 21 Failed To Advance.. Check Qxxx.x French'
  201 = 'Clamp Cylinder A1 Failed to Return... Check Q1.1...' | German: 'S3 201 Row 21 Failed To Return.. Check Qxxx.x German' | French: 'S3 201 Row 21 Failed To Return.. Check Qxxx.x French'
  202 = 'Clamp Cylinder A1 Lost Advanced... Check I1.0...' | German: 'S3 202 Row 21 Lost Advance Position... Check Ixxx.x German' | French: 'S3 202 Row 21 Lost Advance Position... Check Ixxx.x French'
  203 = 'Clamp Cylinder A1 Lost Returned... Check I1.1...' | German: 'S3 203 Row 21 Lost Return Position... Check Ixxx.x German' | French: 'S3 203 Row 21 Lost Return Position... Check Ixxx.x French'
  204 = 'Clamp Cylinder A1 Switch Fault... Check I1.0, I1.1...' | German: 'S3 204 Row 21 Switch Fault... Check Ixxx.x / Ixxx.x German' | French: 'S3 204 Row 21 Switch Fault... Check Ixxx.x / Ixxx.x French'
  205 = 'Spare' | German: 'S3 205 Row 21 Spare Message German' | French: 'S3 205 Row 21 Spare Message French'
  206 = 'Spare' | German: 'S3 206 Row 21 Spare Message German' | French: 'S3 206 Row 21 Spare Message French'
  207 = 'Spare' | German: 'S3 207 Row 21 Spare Message German' | French: 'S3 207 Row 21 Spare Message French'
  208 = 'Spare' | German: 'S3 208 Row 21 Spare Message German' | French: 'S3 208 Row 21 Spare Message French'
  209 = 'Spare' | German: 'S3 209 Row 21 Spare Message German' | French: 'S3 209 Row 21 Spare Message French'
  210 = 'Clamp Cylinder A1 Failed to Advance... Check Q1.0...' | German: 'S3 210 Row 22 Failed To Advance.. Check Qxxx.x German' | French: 'S3 210 Row 22 Failed To Advance.. Check Qxxx.x French'
  211 = 'Clamp Cylinder A1 Failed to Return... Check Q1.1...' | German: 'S3 211 Row 22 Failed To Return.. Check Qxxx.x German' | French: 'S3 211 Row 22 Failed To Return.. Check Qxxx.x French'
  212 = 'Clamp Cylinder A1 Lost Advanced... Check I1.0...' | German: 'S3 212 Row 22 Lost Advance Position... Check Ixxx.x German' | French: 'S3 212 Row 22 Lost Advance Position... Check Ixxx.x French'
  213 = 'Clamp Cylinder A1 Lost Returned... Check I1.1...' | German: 'S3 213 Row 22 Lost Return Position... Check Ixxx.x German' | French: 'S3 213 Row 22 Lost Return Position... Check Ixxx.x French'
  214 = 'Clamp Cylinder A1 Switch Fault... Check I1.0, I1.1...' | German: 'S3 214 Row 22 Switch Fault... Check Ixxx.x / Ixxx.x German' | French: 'S3 214 Row 22 Switch Fault... Check Ixxx.x / Ixxx.x French'
  215 = 'Spare' | German: 'S3 215 Row 22 Spare Message German' | French: 'S3 215 Row 22 Spare Message French'
  216 = 'Spare' | German: 'S3 216 Row 22 Spare Message German' | French: 'S3 216 Row 22 Spare Message French'
  217 = 'Spare' | German: 'S3 217 Row 22 Spare Message German' | French: 'S3 217 Row 22 Spare Message French'
  218 = 'Spare' | German: 'S3 218 Row 22 Spare Message German' | French: 'S3 218 Row 22 Spare Message French'
  219 = 'Spare' | German: 'S3 219 Row 22 Spare Message German' | French: 'S3 219 Row 22 Spare Message French'
  220 = 'Clamp Cylinder A1 Failed to Advance... Check Q1.0...' | German: 'S3 220 Row 23 Failed To Advance.. Check Qxxx.x German' | French: 'S3 220 Row 23 Failed To Advance.. Check Qxxx.x French'
  221 = 'Clamp Cylinder A1 Failed to Return... Check Q1.1...' | German: 'S3 221 Row 23 Failed To Return.. Check Qxxx.x German' | French: 'S3 221 Row 23 Failed To Return.. Check Qxxx.x French'
  222 = 'Clamp Cylinder A1 Lost Advanced... Check I1.0...' | German: 'S3 222 Row 23 Lost Advance Position... Check Ixxx.x German' | French: 'S3 222 Row 23 Lost Advance Position... Check Ixxx.x French'
  223 = 'Clamp Cylinder A1 Lost Returned... Check I1.1...' | German: 'S3 223 Row 23 Lost Return Position... Check Ixxx.x German' | French: 'S3 223 Row 23 Lost Return Position... Check Ixxx.x French'
  224 = 'Clamp Cylinder A1 Switch Fault... Check I1.0, I1.1...' | German: 'S3 224 Row 23 Switch Fault... Check Ixxx.x / Ixxx.x German' | French: 'S3 224 Row 23 Switch Fault... Check Ixxx.x / Ixxx.x French'
  225 = 'Spare' | German: 'S3 225 Row 23 Spare Message German' | French: 'S3 225 Row 23 Spare Message French'
  226 = 'Spare' | German: 'S3 226 Row 23 Spare Message German' | French: 'S3 226 Row 23 Spare Message French'
  227 = 'Spare' | German: 'S3 227 Row 23 Spare Message German' | French: 'S3 227 Row 23 Spare Message French'
  228 = 'Spare' | German: 'S3 228 Row 23 Spare Message German' | French: 'S3 228 Row 23 Spare Message French'
  229 = 'Spare' | German: 'S3 229 Row 23 Spare Message German' | French: 'S3 229 Row 23 Spare Message French'
  230 = 'Clamp Cylinder A1 Failed to Advance... Check Q1.0...' | German: 'S3 230 Row 24 Failed To Advance.. Check Qxxx.x German' | French: 'S3 230 Row 24 Failed To Advance.. Check Qxxx.x French'
  231 = 'Clamp Cylinder A1 Failed to Return... Check Q1.1...' | German: 'S3 231 Row 24 Failed To Return.. Check Qxxx.x German' | French: 'S3 231 Row 24 Failed To Return.. Check Qxxx.x French'
  232 = 'Clamp Cylinder A1 Lost Advanced... Check I1.0...' | German: 'S3 232 Row 24 Lost Advance Position... Check Ixxx.x German' | French: 'S3 232 Row 24 Lost Advance Position... Check Ixxx.x French'
  233 = 'Clamp Cylinder A1 Lost Returned... Check I1.1...' | German: 'S3 233 Row 24 Lost Return Position... Check Ixxx.x German' | French: 'S3 233 Row 24 Lost Return Position... Check Ixxx.x French'
  234 = 'Clamp Cylinder A1 Switch Fault... Check I1.0, I1.1...' | German: 'S3 234 Row 24 Switch Fault... Check Ixxx.x / Ixxx.x German' | French: 'S3 234 Row 24 Switch Fault... Check Ixxx.x / Ixxx.x French'
  235 = 'Spare' | German: 'S3 235 Row 24 Spare Message German' | French: 'S3 235 Row 24 Spare Message French'
  236 = 'Spare' | German: 'S3 236 Row 24 Spare Message German' | French: 'S3 236 Row 24 Spare Message French'
  237 = 'Spare' | German: 'S3 237 Row 24 Spare Message German' | French: 'S3 237 Row 24 Spare Message French'
  238 = 'Spare' | German: 'S3 238 Row 24 Spare Message German' | French: 'S3 238 Row 24 Spare Message French'
  239 = 'Spare' | German: 'S3 239 Row 24 Spare Message German' | French: 'S3 239 Row 24 Spare Message French'
  240 = 'Clamp Cylinder A1 Failed to Advance... Check Q1.0...' | German: 'S3 240 Row 25 Failed To Advance.. Check Qxxx.x German' | French: 'S3 240 Row 25 Failed To Advance.. Check Qxxx.x French'
  241 = 'Clamp Cylinder A1 Failed to Return... Check Q1.1...' | German: 'S3 241 Row 25 Failed To Return.. Check Qxxx.x German' | French: 'S3 241 Row 25 Failed To Return.. Check Qxxx.x French'
  242 = 'Clamp Cylinder A1 Lost Advanced... Check I1.0...' | German: 'S3 242 Row 25 Lost Advance Position... Check Ixxx.x German' | French: 'S3 242 Row 25 Lost Advance Position... Check Ixxx.x French'
  243 = 'Clamp Cylinder A1 Lost Returned... Check I1.1...' | German: 'S3 243 Row 25 Lost Return Position... Check Ixxx.x German' | French: 'S3 243 Row 25 Lost Return Position... Check Ixxx.x French'
  244 = 'Clamp Cylinder A1 Switch Fault... Check I1.0, I1.1...' | German: 'S3 244 Row 25 Switch Fault... Check Ixxx.x / Ixxx.x German' | French: 'S3 244 Row 25 Switch Fault... Check Ixxx.x / Ixxx.x French'
  245 = 'Spare' | German: 'S3 245 Row 25 Spare Message German' | French: 'S3 245 Row 25 Spare Message French'
  246 = 'Spare' | German: 'S3 246 Row 25 Spare Message German' | French: 'S3 246 Row 25 Spare Message French'
  247 = 'Spare' | German: 'S3 247 Row 25 Spare Message German' | French: 'S3 247 Row 25 Spare Message French'
  248 = 'Spare' | German: 'S3 248 Row 25 Spare Message German' | French: 'S3 248 Row 25 Spare Message French'
  249 = 'Spare' | German: 'S3 249 Row 25 Spare Message German' | French: 'S3 249 Row 25 Spare Message French'
  250 = 'Clamp Cylinder A1 Failed to Advance... Check Q1.0...' | German: 'S3 250 Row 26 Failed To Advance.. Check Qxxx.x German' | French: 'S3 250 Row 26 Failed To Advance.. Check Qxxx.x French'
  251 = 'Clamp Cylinder A1 Failed to Return... Check Q1.1...' | German: 'S3 251 Row 26 Failed To Return.. Check Qxxx.x German' | French: 'S3 251 Row 26 Failed To Return.. Check Qxxx.x French'
  252 = 'Clamp Cylinder A1 Lost Advanced... Check I1.0...' | German: 'S3 252 Row 26 Lost Advance Position... Check Ixxx.x German' | French: 'S3 252 Row 26 Lost Advance Position... Check Ixxx.x French'
  253 = 'Clamp Cylinder A1 Lost Returned... Check I1.1...' | German: 'S3 253 Row 26 Lost Return Position... Check Ixxx.x German' | French: 'S3 253 Row 26 Lost Return Position... Check Ixxx.x French'
  254 = 'Clamp Cylinder A1 Switch Fault... Check I1.0, I1.1...' | German: 'S3 254 Row 26 Switch Fault... Check Ixxx.x / Ixxx.x German' | French: 'S3 254 Row 26 Switch Fault... Check Ixxx.x / Ixxx.x French'
  255 = 'Spare' | German: 'S3 255 Row 26 Spare Message German' | French: 'S3 255 Row 26 Spare Message French'
  256 = 'Spare' | German: 'S3 256 Row 26 Spare Message German' | French: 'S3 256 Row 26 Spare Message French'
  257 = 'Spare' | German: 'S3 257 Row 26 Spare Message German' | French: 'S3 257 Row 26 Spare Message French'
  258 = 'Spare' | German: 'S3 258 Row 26 Spare Message German' | French: 'S3 258 Row 26 Spare Message French'
  259 = 'Spare' | German: 'S3 259 Row 26 Spare Message German' | French: 'S3 259 Row 26 Spare Message French'
  260 = 'Clamp Cylinder A1 Failed to Advance... Check Q1.0...' | German: 'S3 260 Row 27 Failed To Advance.. Check Qxxx.x German' | French: 'S3 260 Row 27 Failed To Advance.. Check Qxxx.x French'
  261 = 'Clamp Cylinder A1 Failed to Return... Check Q1.1...' | German: 'S3 261 Row 27 Failed To Return.. Check Qxxx.x German' | French: 'S3 261 Row 27 Failed To Return.. Check Qxxx.x French'
  262 = 'Clamp Cylinder A1 Lost Advanced... Check I1.0...' | German: 'S3 262 Row 27 Lost Advance Position... Check Ixxx.x German' | French: 'S3 262 Row 27 Lost Advance Position... Check Ixxx.x French'
  263 = 'Clamp Cylinder A1 Lost Returned... Check I1.1...' | German: 'S3 263 Row 27 Lost Return Position... Check Ixxx.x German' | French: 'S3 263 Row 27 Lost Return Position... Check Ixxx.x French'
  264 = 'Clamp Cylinder A1 Switch Fault... Check I1.0, I1.1...' | German: 'S3 264 Row 27 Switch Fault... Check Ixxx.x / Ixxx.x German' | French: 'S3 264 Row 27 Switch Fault... Check Ixxx.x / Ixxx.x French'
  265 = 'Spare' | German: 'S3 265 Row 27 Spare Message German' | French: 'S3 265 Row 27 Spare Message French'
  266 = 'Spare' | German: 'S3 266 Row 27 Spare Message German' | French: 'S3 266 Row 27 Spare Message French'
  267 = 'Spare' | German: 'S3 267 Row 27 Spare Message German' | French: 'S3 267 Row 27 Spare Message French'
  268 = 'Spare' | German: 'S3 268 Row 27 Spare Message German' | French: 'S3 268 Row 27 Spare Message French'
  269 = 'Spare' | German: 'S3 269 Row 27 Spare Message German' | French: 'S3 269 Row 27 Spare Message French'
  270 = 'Clamp Cylinder A1 Failed to Advance... Check Q1.0...' | German: 'S3 270 Row 28 Failed To Advance.. Check Qxxx.x German' | French: 'S3 270 Row 28 Failed To Advance.. Check Qxxx.x French'
  271 = 'Clamp Cylinder A1 Failed to Return... Check Q1.1...' | German: 'S3 271 Row 28 Failed To Return.. Check Qxxx.x German' | French: 'S3 271 Row 28 Failed To Return.. Check Qxxx.x French'
  272 = 'Clamp Cylinder A1 Lost Advanced... Check I1.0...' | German: 'S3 272 Row 28 Lost Advance Position... Check Ixxx.x German' | French: 'S3 272 Row 28 Lost Advance Position... Check Ixxx.x French'
  273 = 'Clamp Cylinder A1 Lost Returned... Check I1.1...' | German: 'S3 273 Row 28 Lost Return Position... Check Ixxx.x German' | French: 'S3 273 Row 28 Lost Return Position... Check Ixxx.x French'
  274 = 'Clamp Cylinder A1 Switch Fault... Check I1.0, I1.1...' | German: 'S3 274 Row 28 Switch Fault... Check Ixxx.x / Ixxx.x German' | French: 'S3 274 Row 28 Switch Fault... Check Ixxx.x / Ixxx.x French'
  275 = 'Spare' | German: 'S3 275 Row 28 Spare Message German' | French: 'S3 275 Row 28 Spare Message French'
  276 = 'Spare' | German: 'S3 276 Row 28 Spare Message German' | French: 'S3 276 Row 28 Spare Message French'
  277 = 'Spare' | German: 'S3 277 Row 28 Spare Message German' | French: 'S3 277 Row 28 Spare Message French'
  278 = 'Spare' | German: 'S3 278 Row 28 Spare Message German' | French: 'S3 278 Row 28 Spare Message French'
  279 = 'Spare' | German: 'S3 279 Row 28 Spare Message German' | French: 'S3 279 Row 28 Spare Message French'
  280 = 'Clamp Cylinder A1 Failed to Advance... Check Q1.0...' | German: 'S3 280 Row 29 Failed To Advance.. Check Qxxx.x German' | French: 'S3 280 Row 29 Failed To Advance.. Check Qxxx.x French'
  281 = 'Clamp Cylinder A1 Failed to Return... Check Q1.1...' | German: 'S3 281 Row 29 Failed To Return.. Check Qxxx.x German' | French: 'S3 281 Row 29 Failed To Return.. Check Qxxx.x French'
  282 = 'Clamp Cylinder A1 Lost Advanced... Check I1.0...' | German: 'S3 282 Row 29 Lost Advance Position... Check Ixxx.x German' | French: 'S3 282 Row 29 Lost Advance Position... Check Ixxx.x French'
  283 = 'Clamp Cylinder A1 Lost Returned... Check I1.1...' | German: 'S3 283 Row 29 Lost Return Position... Check Ixxx.x German' | French: 'S3 283 Row 29 Lost Return Position... Check Ixxx.x French'
  284 = 'Clamp Cylinder A1 Switch Fault... Check I1.0, I1.1...' | German: 'S3 284 Row 29 Switch Fault... Check Ixxx.x / Ixxx.x German' | French: 'S3 284 Row 29 Switch Fault... Check Ixxx.x / Ixxx.x French'
  285 = 'Spare' | German: 'S3 285 Row 29 Spare Message German' | French: 'S3 285 Row 29 Spare Message French'
  286 = 'Spare' | German: 'S3 286 Row 29 Spare Message German' | French: 'S3 286 Row 29 Spare Message French'
  287 = 'Spare' | German: 'S3 287 Row 29 Spare Message German' | French: 'S3 287 Row 29 Spare Message French'
  288 = 'Spare' | German: 'S3 288 Row 29 Spare Message German' | French: 'S3 288 Row 29 Spare Message French'
  289 = 'Spare' | German: 'S3 289 Row 29 Spare Message German' | French: 'S3 289 Row 29 Spare Message French'
  290 = 'Clamp Cylinder A1 Failed to Advance... Check Q1.0...' | German: 'S3 290 Row 30 Failed To Advance.. Check Qxxx.x German' | French: 'S3 290 Row 30 Failed To Advance.. Check Qxxx.x French'
  291 = 'Clamp Cylinder A1 Failed to Return... Check Q1.1...' | German: 'S3 291 Row 30 Failed To Return.. Check Qxxx.x German' | French: 'S3 291 Row 30 Failed To Return.. Check Qxxx.x French'
  292 = 'Clamp Cylinder A1 Lost Advanced... Check I1.0...' | German: 'S3 292 Row 30 Lost Advance Position... Check Ixxx.x German' | French: 'S3 292 Row 30 Lost Advance Position... Check Ixxx.x French'
  293 = 'Clamp Cylinder A1 Lost Returned... Check I1.1...' | German: 'S3 293 Row 30 Lost Return Position... Check Ixxx.x German' | French: 'S3 293 Row 30 Lost Return Position... Check Ixxx.x French'
  294 = 'Clamp Cylinder A1 Switch Fault... Check I1.0, I1.1...' | German: 'S3 294 Row 30 Switch Fault... Check Ixxx.x / Ixxx.x German' | French: 'S3 294 Row 30 Switch Fault... Check Ixxx.x / Ixxx.x French'
  295 = 'Spare' | German: 'S3 295 Row 30 Spare Message German' | French: 'S3 295 Row 30 Spare Message French'
  296 = 'Spare' | German: 'S3 296 Row 30 Spare Message German' | French: 'S3 296 Row 30 Spare Message French'
  297 = 'Spare' | German: 'S3 297 Row 30 Spare Message German' | French: 'S3 297 Row 30 Spare Message French'
  298 = 'Spare' | German: 'S3 298 Row 30 Spare Message German' | French: 'S3 298 Row 30 Spare Message French'
  299 = 'Spare' | German: 'S3 299 Row 30 Spare Message German' | French: 'S3 299 Row 30 Spare Message French'
  300 = 'Clamp Cylinder A1 Failed to Advance... Check Q1.0...' | German: 'S3 300 Row 31 Failed To Advance.. Check Qxxx.x German' | French: 'S3 300 Row 31 Failed To Advance.. Check Qxxx.x French'
  301 = 'Clamp Cylinder A1 Failed to Return... Check Q1.1...' | German: 'S3 301 Row 31 Failed To Return.. Check Qxxx.x German' | French: 'S3 301 Row 31 Failed To Return.. Check Qxxx.x French'
  302 = 'Clamp Cylinder A1 Lost Advanced... Check I1.0...' | German: 'S3 302 Row 31 Lost Advance Position... Check Ixxx.x German' | French: 'S3 302 Row 31 Lost Advance Position... Check Ixxx.x French'
  303 = 'Clamp Cylinder A1 Lost Returned... Check I1.1...' | German: 'S3 303 Row 31 Lost Return Position... Check Ixxx.x German' | French: 'S3 303 Row 31 Lost Return Position... Check Ixxx.x French'
  304 = 'Clamp Cylinder A1 Switch Fault... Check I1.0, I1.1...' | German: 'S3 304 Row 31 Switch Fault... Check Ixxx.x / Ixxx.x German' | French: 'S3 304 Row 31 Switch Fault... Check Ixxx.x / Ixxx.x French'
  305 = 'Spare' | German: 'S3 305 Row 31 Spare Message German' | French: 'S3 305 Row 31 Spare Message French'
  306 = 'Spare' | German: 'S3 306 Row 31 Spare Message German' | French: 'S3 306 Row 31 Spare Message French'
  307 = 'Spare' | German: 'S3 307 Row 31 Spare Message German' | French: 'S3 307 Row 31 Spare Message French'
  308 = 'Spare' | German: 'S3 308 Row 31 Spare Message German' | French: 'S3 308 Row 31 Spare Message French'
  309 = 'Spare' | German: 'S3 309 Row 31 Spare Message German' | French: 'S3 309 Row 31 Spare Message French'
  310 = 'Clamp Cylinder A1 Failed to Advance... Check Q1.0...' | German: 'S3 310 Row 32 Failed To Advance.. Check Qxxx.x German' | French: 'S3 310 Row 32 Failed To Advance.. Check Qxxx.x French'
  311 = 'Clamp Cylinder A1 Failed to Return... Check Q1.1...' | German: 'S3 311 Row 32 Failed To Return.. Check Qxxx.x German' | French: 'S3 311 Row 32 Failed To Return.. Check Qxxx.x French'
  312 = 'Clamp Cylinder A1 Lost Advanced... Check I1.0...' | German: 'S3 312 Row 32 Lost Advance Position... Check Ixxx.x German' | French: 'S3 312 Row 32 Lost Advance Position... Check Ixxx.x French'
  313 = 'Clamp Cylinder A1 Lost Returned... Check I1.1...' | German: 'S3 313 Row 32 Lost Return Position... Check Ixxx.x German' | French: 'S3 313 Row 32 Lost Return Position... Check Ixxx.x French'
  314 = 'Clamp Cylinder A1 Switch Fault... Check I1.0, I1.1...' | German: 'S3 314 Row 32 Switch Fault... Check Ixxx.x / Ixxx.x German' | French: 'S3 314 Row 32 Switch Fault... Check Ixxx.x / Ixxx.x French'
  315 = 'Spare' | German: 'S3 315 Row 32 Spare Message German' | French: 'S3 315 Row 32 Spare Message French'
  316 = 'Spare' | German: 'S3 316 Row 32 Spare Message German' | French: 'S3 316 Row 32 Spare Message French'
  317 = 'Spare' | German: 'S3 317 Row 32 Spare Message German' | French: 'S3 317 Row 32 Spare Message French'
  318 = 'Spare' | German: 'S3 318 Row 32 Spare Message German' | French: 'S3 318 Row 32 Spare Message French'
  319 = 'Spare' | German: 'S3 319 Row 32 Spare Message German' | French: 'S3 319 Row 32 Spare Message French'
  320 = 'Clamp Cylinder A1 Failed to Advance... Check Q1.0...' | German: 'S3 320 Row 33 Failed To Advance.. Check Qxxx.x German' | French: 'S3 320 Row 33 Failed To Advance.. Check Qxxx.x French'
  321 = 'Clamp Cylinder A1 Failed to Return... Check Q1.1...' | German: 'S3 321 Row 33 Failed To Return.. Check Qxxx.x German' | French: 'S3 321 Row 33 Failed To Return.. Check Qxxx.x French'
  322 = 'Clamp Cylinder A1 Lost Advanced... Check I1.0...' | German: 'S3 322 Row 33 Lost Advance Position... Check Ixxx.x German' | French: 'S3 322 Row 33 Lost Advance Position... Check Ixxx.x French'
  323 = 'Clamp Cylinder A1 Lost Returned... Check I1.1...' | German: 'S3 323 Row 33 Lost Return Position... Check Ixxx.x German' | French: 'S3 323 Row 33 Lost Return Position... Check Ixxx.x French'
  324 = 'Clamp Cylinder A1 Switch Fault... Check I1.0, I1.1...' | German: 'S3 324 Row 33 Switch Fault... Check Ixxx.x / Ixxx.x German' | French: 'S3 324 Row 33 Switch Fault... Check Ixxx.x / Ixxx.x French'
  325 = 'Spare' | German: 'S3 325 Row 33 Spare Message German' | French: 'S3 325 Row 33 Spare Message French'
  326 = 'Spare' | German: 'S3 326 Row 33 Spare Message German' | French: 'S3 326 Row 33 Spare Message French'
  327 = 'Spare' | German: 'S3 327 Row 33 Spare Message German' | French: 'S3 327 Row 33 Spare Message French'
  328 = 'Spare' | German: 'S3 328 Row 33 Spare Message German' | French: 'S3 328 Row 33 Spare Message French'
  329 = 'Spare' | German: 'S3 329 Row 33 Spare Message German' | French: 'S3 329 Row 33 Spare Message French'
  330 = 'Clamp Cylinder A1 Failed to Advance... Check Q1.0...' | German: 'S3 330 Row 34 Failed To Advance.. Check Qxxx.x German' | French: 'S3 330 Row 34 Failed To Advance.. Check Qxxx.x French'
  331 = 'Clamp Cylinder A1 Failed to Return... Check Q1.1...' | German: 'S3 331 Row 34 Failed To Return.. Check Qxxx.x German' | French: 'S3 331 Row 34 Failed To Return.. Check Qxxx.x French'
  332 = 'Clamp Cylinder A1 Lost Advanced... Check I1.0...' | German: 'S3 332 Row 34 Lost Advance Position... Check Ixxx.x German' | French: 'S3 332 Row 34 Lost Advance Position... Check Ixxx.x French'
  333 = 'Clamp Cylinder A1 Lost Returned... Check I1.1...' | German: 'S3 333 Row 34 Lost Return Position... Check Ixxx.x German' | French: 'S3 333 Row 34 Lost Return Position... Check Ixxx.x French'
  334 = 'Clamp Cylinder A1 Switch Fault... Check I1.0, I1.1...' | German: 'S3 334 Row 34 Switch Fault... Check Ixxx.x / Ixxx.x German' | French: 'S3 334 Row 34 Switch Fault... Check Ixxx.x / Ixxx.x French'
  335 = 'Spare' | German: 'S3 335 Row 34 Spare Message German' | French: 'S3 335 Row 34 Spare Message French'
  336 = 'Spare' | German: 'S3 336 Row 34 Spare Message German' | French: 'S3 336 Row 34 Spare Message French'
  337 = 'Spare' | German: 'S3 337 Row 34 Spare Message German' | French: 'S3 337 Row 34 Spare Message French'
  338 = 'Spare' | German: 'S3 338 Row 34 Spare Message German' | French: 'S3 338 Row 34 Spare Message French'
  339 = 'Spare' | German: 'S3 339 Row 34 Spare Message German' | French: 'S3 339 Row 34 Spare Message French'
  340 = 'Clamp Cylinder A1 Failed to Advance... Check Q1.0...' | German: 'S3 340 Row 35 Failed To Advance.. Check Qxxx.x German' | French: 'S3 340 Row 35 Failed To Advance.. Check Qxxx.x French'
  341 = 'Clamp Cylinder A1 Failed to Return... Check Q1.1...' | German: 'S3 341 Row 35 Failed To Return.. Check Qxxx.x German' | French: 'S3 341 Row 35 Failed To Return.. Check Qxxx.x French'
  342 = 'Clamp Cylinder A1 Lost Advanced... Check I1.0...' | German: 'S3 342 Row 35 Lost Advance Position... Check Ixxx.x German' | French: 'S3 342 Row 35 Lost Advance Position... Check Ixxx.x French'
  343 = 'Clamp Cylinder A1 Lost Returned... Check I1.1...' | German: 'S3 343 Row 35 Lost Return Position... Check Ixxx.x German' | French: 'S3 343 Row 35 Lost Return Position... Check Ixxx.x French'
  344 = 'Clamp Cylinder A1 Switch Fault... Check I1.0, I1.1...' | German: 'S3 344 Row 35 Switch Fault... Check Ixxx.x / Ixxx.x German' | French: 'S3 344 Row 35 Switch Fault... Check Ixxx.x / Ixxx.x French'
  345 = 'Spare' | German: 'S3 345 Row 35 Spare Message German' | French: 'S3 345 Row 35 Spare Message French'
  346 = 'Spare' | German: 'S3 346 Row 35 Spare Message German' | French: 'S3 346 Row 35 Spare Message French'
  347 = 'Spare' | German: 'S3 347 Row 35 Spare Message German' | French: 'S3 347 Row 35 Spare Message French'
  348 = 'Spare' | German: 'S3 348 Row 35 Spare Message German' | French: 'S3 348 Row 35 Spare Message French'
  349 = 'Spare' | German: 'S3 349 Row 35 Spare Message German' | French: 'S3 349 Row 35 Spare Message French'
  350 = 'Clamp Cylinder A1 Failed to Advance... Check Q1.0...' | German: 'S3 350 Row 36 Failed To Advance.. Check Qxxx.x German' | French: 'S3 350 Row 36 Failed To Advance.. Check Qxxx.x French'
  351 = 'Clamp Cylinder A1 Failed to Return... Check Q1.1...' | German: 'S3 351 Row 36 Failed To Return.. Check Qxxx.x German' | French: 'S3 351 Row 36 Failed To Return.. Check Qxxx.x French'
  352 = 'Clamp Cylinder A1 Lost Advanced... Check I1.0...' | German: 'S3 352 Row 36 Lost Advance Position... Check Ixxx.x German' | French: 'S3 352 Row 36 Lost Advance Position... Check Ixxx.x French'
  353 = 'Clamp Cylinder A1 Lost Returned... Check I1.1...' | German: 'S3 353 Row 36 Lost Return Position... Check Ixxx.x German' | French: 'S3 353 Row 36 Lost Return Position... Check Ixxx.x French'
  354 = 'Clamp Cylinder A1 Switch Fault... Check I1.0, I1.1...' | German: 'S3 354 Row 36 Switch Fault... Check Ixxx.x / Ixxx.x German' | French: 'S3 354 Row 36 Switch Fault... Check Ixxx.x / Ixxx.x French'
  355 = 'Spare' | German: 'S3 355 Row 36 Spare Message German' | French: 'S3 355 Row 36 Spare Message French'
  356 = 'Spare' | German: 'S3 356 Row 36 Spare Message German' | French: 'S3 356 Row 36 Spare Message French'
  357 = 'Spare' | German: 'S3 357 Row 36 Spare Message German' | French: 'S3 357 Row 36 Spare Message French'
  358 = 'Spare' | German: 'S3 358 Row 36 Spare Message German' | French: 'S3 358 Row 36 Spare Message French'
  359 = 'Spare' | German: 'S3 359 Row 36 Spare Message German' | French: 'S3 359 Row 36 Spare Message French'
  360 = 'Clamp Cylinder A1 Failed to Advance... Check Q1.0...' | German: 'S3 360 Row 37 Failed To Advance.. Check Qxxx.x German' | French: 'S3 360 Row 37 Failed To Advance.. Check Qxxx.x French'
  361 = 'Clamp Cylinder A1 Failed to Return... Check Q1.1...' | German: 'S3 361 Row 37 Failed To Return.. Check Qxxx.x German' | French: 'S3 361 Row 37 Failed To Return.. Check Qxxx.x French'
  362 = 'Clamp Cylinder A1 Lost Advanced... Check I1.0...' | German: 'S3 362 Row 37 Lost Advance Position... Check Ixxx.x German' | French: 'S3 362 Row 37 Lost Advance Position... Check Ixxx.x French'
  363 = 'Clamp Cylinder A1 Lost Returned... Check I1.1...' | German: 'S3 363 Row 37 Lost Return Position... Check Ixxx.x German' | French: 'S3 363 Row 37 Lost Return Position... Check Ixxx.x French'
  364 = 'Clamp Cylinder A1 Switch Fault... Check I1.0, I1.1...' | German: 'S3 364 Row 37 Switch Fault... Check Ixxx.x / Ixxx.x German' | French: 'S3 364 Row 37 Switch Fault... Check Ixxx.x / Ixxx.x French'
  365 = 'Spare' | German: 'S3 365 Row 37 Spare Message German' | French: 'S3 365 Row 37 Spare Message French'
  366 = 'Spare' | German: 'S3 366 Row 37 Spare Message German' | French: 'S3 366 Row 37 Spare Message French'
  367 = 'Spare' | German: 'S3 367 Row 37 Spare Message German' | French: 'S3 367 Row 37 Spare Message French'
  368 = 'Spare' | German: 'S3 368 Row 37 Spare Message German' | French: 'S3 368 Row 37 Spare Message French'
  369 = 'Spare' | German: 'S3 369 Row 37 Spare Message German' | French: 'S3 369 Row 37 Spare Message French'
  370 = 'Clamp Cylinder A1 Failed to Advance... Check Q1.0...' | German: 'S3 370 Row 38 Failed To Advance.. Check Qxxx.x German' | French: 'S3 370 Row 38 Failed To Advance.. Check Qxxx.x French'
  371 = 'Clamp Cylinder A1 Failed to Return... Check Q1.1...' | German: 'S3 371 Row 38 Failed To Return.. Check Qxxx.x German' | French: 'S3 371 Row 38 Failed To Return.. Check Qxxx.x French'
  372 = 'Clamp Cylinder A1 Lost Advanced... Check I1.0...' | German: 'S3 372 Row 38 Lost Advance Position... Check Ixxx.x German' | French: 'S3 372 Row 38 Lost Advance Position... Check Ixxx.x French'
  373 = 'Clamp Cylinder A1 Lost Returned... Check I1.1...' | German: 'S3 373 Row 38 Lost Return Position... Check Ixxx.x German' | French: 'S3 373 Row 38 Lost Return Position... Check Ixxx.x French'
  374 = 'Clamp Cylinder A1 Switch Fault... Check I1.0, I1.1...' | German: 'S3 374 Row 38 Switch Fault... Check Ixxx.x / Ixxx.x German' | French: 'S3 374 Row 38 Switch Fault... Check Ixxx.x / Ixxx.x French'
  375 = 'Spare' | German: 'S3 375 Row 38 Spare Message German' | French: 'S3 375 Row 38 Spare Message French'
  376 = 'Spare' | German: 'S3 376 Row 38 Spare Message German' | French: 'S3 376 Row 38 Spare Message French'
  377 = 'Spare' | German: 'S3 377 Row 38 Spare Message German' | French: 'S3 377 Row 38 Spare Message French'
  378 = 'Spare' | German: 'S3 378 Row 38 Spare Message German' | French: 'S3 378 Row 38 Spare Message French'
  379 = 'Spare' | German: 'S3 379 Row 38 Spare Message German' | French: 'S3 379 Row 38 Spare Message French'
  380 = 'Clamp Cylinder A1 Failed to Advance... Check Q1.0...' | German: 'S3 380 Row 39 Failed To Advance.. Check Qxxx.x German' | French: 'S3 380 Row 39 Failed To Advance.. Check Qxxx.x French'
  381 = 'Clamp Cylinder A1 Failed to Return... Check Q1.1...' | German: 'S3 381 Row 39 Failed To Return.. Check Qxxx.x German' | French: 'S3 381 Row 39 Failed To Return.. Check Qxxx.x French'
  382 = 'Clamp Cylinder A1 Lost Advanced... Check I1.0...' | German: 'S3 382 Row 39 Lost Advance Position... Check Ixxx.x German' | French: 'S3 382 Row 39 Lost Advance Position... Check Ixxx.x French'
  383 = 'Clamp Cylinder A1 Lost Returned... Check I1.1...' | German: 'S3 383 Row 39 Lost Return Position... Check Ixxx.x German' | French: 'S3 383 Row 39 Lost Return Position... Check Ixxx.x French'
  384 = 'Clamp Cylinder A1 Switch Fault... Check I1.0, I1.1...' | German: 'S3 384 Row 39 Switch Fault... Check Ixxx.x / Ixxx.x German' | French: 'S3 384 Row 39 Switch Fault... Check Ixxx.x / Ixxx.x French'
  385 = 'Spare' | German: 'S3 385 Row 39 Spare Message German' | French: 'S3 385 Row 39 Spare Message French'
  386 = 'Spare' | German: 'S3 386 Row 39 Spare Message German' | French: 'S3 386 Row 39 Spare Message French'
  387 = 'Spare' | German: 'S3 387 Row 39 Spare Message German' | French: 'S3 387 Row 39 Spare Message French'
  388 = 'Spare' | German: 'S3 388 Row 39 Spare Message German' | French: 'S3 388 Row 39 Spare Message French'
  389 = 'Spare' | German: 'S3 389 Row 39 Spare Message German' | French: 'S3 389 Row 39 Spare Message French'
  390 = 'Clamp Cylinder A1 Failed to Advance... Check Q1.0...' | German: 'S3 390 Row 40 Failed To Advance.. Check Qxxx.x German' | French: 'S3 390 Row 40 Failed To Advance.. Check Qxxx.x French'
  391 = 'Clamp Cylinder A1 Failed to Return... Check Q1.1...' | German: 'S3 391 Row 40 Failed To Return.. Check Qxxx.x German' | French: 'S3 391 Row 40 Failed To Return.. Check Qxxx.x French'
  392 = 'Clamp Cylinder A1 Lost Advanced... Check I1.0...' | German: 'S3 392 Row 40 Lost Advance Position... Check Ixxx.x German' | French: 'S3 392 Row 40 Lost Advance Position... Check Ixxx.x French'
  393 = 'Clamp Cylinder A1 Lost Returned... Check I1.1...' | German: 'S3 393 Row 40 Lost Return Position... Check Ixxx.x German' | French: 'S3 393 Row 40 Lost Return Position... Check Ixxx.x French'
  394 = 'Clamp Cylinder A1 Switch Fault... Check I1.0, I1.1...' | German: 'S3 394 Row 40 Switch Fault... Check Ixxx.x / Ixxx.x German' | French: 'S3 394 Row 40 Switch Fault... Check Ixxx.x / Ixxx.x French'
  395 = 'Spare' | German: 'S3 395 Row 40 Spare Message German' | French: 'S3 395 Row 40 Spare Message French'
  396 = 'Spare' | German: 'S3 396 Row 40 Spare Message German' | French: 'S3 396 Row 40 Spare Message French'
  397 = 'Spare' | German: 'S3 397 Row 40 Spare Message German' | French: 'S3 397 Row 40 Spare Message French'
  398 = 'Spare' | German: 'S3 398 Row 40 Spare Message German' | French: 'S3 398 Row 40 Spare Message French'
  399 = 'Spare' | German: 'S3 399 Row 40 Spare Message German' | French: 'S3 399 Row 40 Spare Message French'
  400 = 'Clamp Cylinder A1 Failed to Advance... Check Q1.0...' | German: 'S3 400 Row 41 Failed To Advance.. Check Qxxx.x German' | French: 'S3 400 Row 41 Failed To Advance.. Check Qxxx.x French'
  401 = 'Clamp Cylinder A1 Failed to Return... Check Q1.1...' | German: 'S3 401 Row 41 Failed To Return.. Check Qxxx.x German' | French: 'S3 401 Row 41 Failed To Return.. Check Qxxx.x French'
  402 = 'Clamp Cylinder A1 Lost Advanced... Check I1.0...' | German: 'S3 402 Row 41 Lost Advance Position... Check Ixxx.x German' | French: 'S3 402 Row 41 Lost Advance Position... Check Ixxx.x French'
  403 = 'Clamp Cylinder A1 Lost Returned... Check I1.1...' | German: 'S3 403 Row 41 Lost Return Position... Check Ixxx.x German' | French: 'S3 403 Row 41 Lost Return Position... Check Ixxx.x French'
  404 = 'Clamp Cylinder A1 Switch Fault... Check I1.0, I1.1...' | German: 'S3 404 Row 41 Switch Fault... Check Ixxx.x / Ixxx.x German' | French: 'S3 404 Row 41 Switch Fault... Check Ixxx.x / Ixxx.x French'
  405 = 'Spare' | German: 'S3 405 Row 41 Spare Message German' | French: 'S3 405 Row 41 Spare Message French'
  406 = 'Spare' | German: 'S3 406 Row 41 Spare Message German' | French: 'S3 406 Row 41 Spare Message French'
  407 = 'Spare' | German: 'S3 407 Row 41 Spare Message German' | French: 'S3 407 Row 41 Spare Message French'
  408 = 'Spare' | German: 'S3 408 Row 41 Spare Message German' | French: 'S3 408 Row 41 Spare Message French'
  409 = 'Spare' | German: 'S3 409 Row 41 Spare Message German' | French: 'S3 409 Row 41 Spare Message French'
  410 = 'Clamp Cylinder A1 Failed to Advance... Check Q1.0...' | German: 'S3 410 Row 42 Failed To Advance.. Check Qxxx.x German' | French: 'S3 410 Row 42 Failed To Advance.. Check Qxxx.x French'
  411 = 'Clamp Cylinder A1 Failed to Return... Check Q1.1...' | German: 'S3 411 Row 42 Failed To Return.. Check Qxxx.x German' | French: 'S3 411 Row 42 Failed To Return.. Check Qxxx.x French'
  412 = 'Clamp Cylinder A1 Lost Advanced... Check I1.0...' | German: 'S3 412 Row 42 Lost Advance Position... Check Ixxx.x German' | French: 'S3 412 Row 42 Lost Advance Position... Check Ixxx.x French'
  413 = 'Clamp Cylinder A1 Lost Returned... Check I1.1...' | German: 'S3 413 Row 42 Lost Return Position... Check Ixxx.x German' | French: 'S3 413 Row 42 Lost Return Position... Check Ixxx.x French'
  414 = 'Clamp Cylinder A1 Switch Fault... Check I1.0, I1.1...' | German: 'S3 414 Row 42 Switch Fault... Check Ixxx.x / Ixxx.x German' | French: 'S3 414 Row 42 Switch Fault... Check Ixxx.x / Ixxx.x French'
  415 = 'Spare' | German: 'S3 415 Row 42 Spare Message German' | French: 'S3 415 Row 42 Spare Message French'
  416 = 'Spare' | German: 'S3 416 Row 42 Spare Message German' | French: 'S3 416 Row 42 Spare Message French'
  417 = 'Spare' | German: 'S3 417 Row 42 Spare Message German' | French: 'S3 417 Row 42 Spare Message French'
  418 = 'Spare' | German: 'S3 418 Row 42 Spare Message German' | French: 'S3 418 Row 42 Spare Message French'
  419 = 'Spare' | German: 'S3 419 Row 42 Spare Message German' | French: 'S3 419 Row 42 Spare Message French'
  420 = 'Clamp Cylinder A1 Failed to Advance... Check Q1.0...' | German: 'S3 420 Row 43 Failed To Advance.. Check Qxxx.x German' | French: 'S3 420 Row 43 Failed To Advance.. Check Qxxx.x French'
  421 = 'Clamp Cylinder A1 Failed to Return... Check Q1.1...' | German: 'S3 421 Row 43 Failed To Return.. Check Qxxx.x German' | French: 'S3 421 Row 43 Failed To Return.. Check Qxxx.x French'
  422 = 'Clamp Cylinder A1 Lost Advanced... Check I1.0...' | German: 'S3 422 Row 43 Lost Advance Position... Check Ixxx.x German' | French: 'S3 422 Row 43 Lost Advance Position... Check Ixxx.x French'
  423 = 'Clamp Cylinder A1 Lost Returned... Check I1.1...' | German: 'S3 423 Row 43 Lost Return Position... Check Ixxx.x German' | French: 'S3 423 Row 43 Lost Return Position... Check Ixxx.x French'
  424 = 'Clamp Cylinder A1 Switch Fault... Check I1.0, I1.1...' | German: 'S3 424 Row 43 Switch Fault... Check Ixxx.x / Ixxx.x German' | French: 'S3 424 Row 43 Switch Fault... Check Ixxx.x / Ixxx.x French'
  425 = 'Spare' | German: 'S3 425 Row 43 Spare Message German' | French: 'S3 425 Row 43 Spare Message French'
  426 = 'Spare' | German: 'S3 426 Row 43 Spare Message German' | French: 'S3 426 Row 43 Spare Message French'
  427 = 'Spare' | German: 'S3 427 Row 43 Spare Message German' | French: 'S3 427 Row 43 Spare Message French'
  428 = 'Spare' | German: 'S3 428 Row 43 Spare Message German' | French: 'S3 428 Row 43 Spare Message French'
  429 = 'Spare' | German: 'S3 429 Row 43 Spare Message German' | French: 'S3 429 Row 43 Spare Message French'
  430 = 'Clamp Cylinder A1 Failed to Advance... Check Q1.0...' | German: 'S3 430 Row 44 Failed To Advance.. Check Qxxx.x German' | French: 'S3 430 Row 44 Failed To Advance.. Check Qxxx.x French'
  431 = 'Clamp Cylinder A1 Failed to Return... Check Q1.1...' | German: 'S3 431 Row 44 Failed To Return.. Check Qxxx.x German' | French: 'S3 431 Row 44 Failed To Return.. Check Qxxx.x French'
  432 = 'Clamp Cylinder A1 Lost Advanced... Check I1.0...' | German: 'S3 432 Row 44 Lost Advance Position... Check Ixxx.x German' | French: 'S3 432 Row 44 Lost Advance Position... Check Ixxx.x French'
  433 = 'Clamp Cylinder A1 Lost Returned... Check I1.1...' | German: 'S3 433 Row 44 Lost Return Position... Check Ixxx.x German' | French: 'S3 433 Row 44 Lost Return Position... Check Ixxx.x French'
  434 = 'Clamp Cylinder A1 Switch Fault... Check I1.0, I1.1...' | German: 'S3 434 Row 44 Switch Fault... Check Ixxx.x / Ixxx.x German' | French: 'S3 434 Row 44 Switch Fault... Check Ixxx.x / Ixxx.x French'
  435 = 'Spare' | German: 'S3 435 Row 44 Spare Message German' | French: 'S3 435 Row 44 Spare Message French'
  436 = 'Spare' | German: 'S3 436 Row 44 Spare Message German' | French: 'S3 436 Row 44 Spare Message French'
  437 = 'Spare' | German: 'S3 437 Row 44 Spare Message German' | French: 'S3 437 Row 44 Spare Message French'
  438 = 'Spare' | German: 'S3 438 Row 44 Spare Message German' | French: 'S3 438 Row 44 Spare Message French'
  439 = 'Spare' | German: 'S3 439 Row 44 Spare Message German' | French: 'S3 439 Row 44 Spare Message French'
  440 = 'Clamp Cylinder A1 Failed to Advance... Check Q1.0...' | German: 'S3 440 Row 45 Failed To Advance.. Check Qxxx.x German' | French: 'S3 440 Row 45 Failed To Advance.. Check Qxxx.x French'
  441 = 'Clamp Cylinder A1 Failed to Return... Check Q1.1...' | German: 'S3 441 Row 45 Failed To Return.. Check Qxxx.x German' | French: 'S3 441 Row 45 Failed To Return.. Check Qxxx.x French'
  442 = 'Clamp Cylinder A1 Lost Advanced... Check I1.0...' | German: 'S3 442 Row 45 Lost Advance Position... Check Ixxx.x German' | French: 'S3 442 Row 45 Lost Advance Position... Check Ixxx.x French'
  443 = 'Clamp Cylinder A1 Lost Returned... Check I1.1...' | German: 'S3 443 Row 45 Lost Return Position... Check Ixxx.x German' | French: 'S3 443 Row 45 Lost Return Position... Check Ixxx.x French'
  444 = 'Clamp Cylinder A1 Switch Fault... Check I1.0, I1.1...' | German: 'S3 444 Row 45 Switch Fault... Check Ixxx.x / Ixxx.x German' | French: 'S3 444 Row 45 Switch Fault... Check Ixxx.x / Ixxx.x French'
  445 = 'Spare' | German: 'S3 445 Row 45 Spare Message German' | French: 'S3 445 Row 45 Spare Message French'
  446 = 'Spare' | German: 'S3 446 Row 45 Spare Message German' | French: 'S3 446 Row 45 Spare Message French'
  447 = 'Spare' | German: 'S3 447 Row 45 Spare Message German' | French: 'S3 447 Row 45 Spare Message French'
  448 = 'Spare' | German: 'S3 448 Row 45 Spare Message German' | French: 'S3 448 Row 45 Spare Message French'
  449 = 'Spare' | German: 'S3 449 Row 45 Spare Message German' | French: 'S3 449 Row 45 Spare Message French'
  450 = 'Clamp Cylinder A1 Failed to Advance... Check Q1.0...' | German: 'S3 450 Row 46 Failed To Advance.. Check Qxxx.x German' | French: 'S3 450 Row 46 Failed To Advance.. Check Qxxx.x French'
  451 = 'Clamp Cylinder A1 Failed to Return... Check Q1.1...' | German: 'S3 451 Row 46 Failed To Return.. Check Qxxx.x German' | French: 'S3 451 Row 46 Failed To Return.. Check Qxxx.x French'
  452 = 'Clamp Cylinder A1 Lost Advanced... Check I1.0...' | German: 'S3 452 Row 46 Lost Advance Position... Check Ixxx.x German' | French: 'S3 452 Row 46 Lost Advance Position... Check Ixxx.x French'
  453 = 'Clamp Cylinder A1 Lost Returned... Check I1.1...' | German: 'S3 453 Row 46 Lost Return Position... Check Ixxx.x German' | French: 'S3 453 Row 46 Lost Return Position... Check Ixxx.x French'
  454 = 'Clamp Cylinder A1 Switch Fault... Check I1.0, I1.1...' | German: 'S3 454 Row 46 Switch Fault... Check Ixxx.x / Ixxx.x German' | French: 'S3 454 Row 46 Switch Fault... Check Ixxx.x / Ixxx.x French'
  455 = 'Spare' | German: 'S3 455 Row 46 Spare Message German' | French: 'S3 455 Row 46 Spare Message French'
  456 = 'Spare' | German: 'S3 456 Row 46 Spare Message German' | French: 'S3 456 Row 46 Spare Message French'
  457 = 'Spare' | German: 'S3 457 Row 46 Spare Message German' | French: 'S3 457 Row 46 Spare Message French'
  458 = 'Spare' | German: 'S3 458 Row 46 Spare Message German' | French: 'S3 458 Row 46 Spare Message French'
  459 = 'Spare' | German: 'S3 459 Row 46 Spare Message German' | French: 'S3 459 Row 46 Spare Message French'
  460 = 'Clamp Cylinder A1 Failed to Advance... Check Q1.0...' | German: 'S3 460 Row 47 Failed To Advance.. Check Qxxx.x German' | French: 'S3 460 Row 47 Failed To Advance.. Check Qxxx.x French'
  461 = 'Clamp Cylinder A1 Failed to Return... Check Q1.1...' | German: 'S3 461 Row 47 Failed To Return.. Check Qxxx.x German' | French: 'S3 461 Row 47 Failed To Return.. Check Qxxx.x French'
  462 = 'Clamp Cylinder A1 Lost Advanced... Check I1.0...' | German: 'S3 462 Row 47 Lost Advance Position... Check Ixxx.x German' | French: 'S3 462 Row 47 Lost Advance Position... Check Ixxx.x French'
  463 = 'Clamp Cylinder A1 Lost Returned... Check I1.1...' | German: 'S3 463 Row 47 Lost Return Position... Check Ixxx.x German' | French: 'S3 463 Row 47 Lost Return Position... Check Ixxx.x French'
  464 = 'Clamp Cylinder A1 Switch Fault... Check I1.0, I1.1...' | German: 'S3 464 Row 47 Switch Fault... Check Ixxx.x / Ixxx.x German' | French: 'S3 464 Row 47 Switch Fault... Check Ixxx.x / Ixxx.x French'
  465 = 'Spare' | German: 'S3 465 Row 47 Spare Message German' | French: 'S3 465 Row 47 Spare Message French'
  466 = 'Spare' | German: 'S3 466 Row 47 Spare Message German' | French: 'S3 466 Row 47 Spare Message French'
  467 = 'Spare' | German: 'S3 467 Row 47 Spare Message German' | French: 'S3 467 Row 47 Spare Message French'
  468 = 'Spare' | German: 'S3 468 Row 47 Spare Message German' | French: 'S3 468 Row 47 Spare Message French'
  469 = 'Spare' | German: 'S3 469 Row 47 Spare Message German' | French: 'S3 469 Row 47 Spare Message French'
  470 = 'Clamp Cylinder A1 Failed to Advance... Check Q1.0...' | German: 'S3 470 Row 48 Failed To Advance.. Check Qxxx.x German' | French: 'S3 470 Row 48 Failed To Advance.. Check Qxxx.x French'
  471 = 'Clamp Cylinder A1 Failed to Return... Check Q1.1...' | German: 'S3 471 Row 48 Failed To Return.. Check Qxxx.x German' | French: 'S3 471 Row 48 Failed To Return.. Check Qxxx.x French'
  472 = 'Clamp Cylinder A1 Lost Advanced... Check I1.0...' | German: 'S3 472 Row 48 Lost Advance Position... Check Ixxx.x German' | French: 'S3 472 Row 48 Lost Advance Position... Check Ixxx.x French'
  473 = 'Clamp Cylinder A1 Lost Returned... Check I1.1...' | German: 'S3 473 Row 48 Lost Return Position... Check Ixxx.x German' | French: 'S3 473 Row 48 Lost Return Position... Check Ixxx.x French'
  474 = 'Clamp Cylinder A1 Switch Fault... Check I1.0, I1.1...' | German: 'S3 474 Row 48 Switch Fault... Check Ixxx.x / Ixxx.x German' | French: 'S3 474 Row 48 Switch Fault... Check Ixxx.x / Ixxx.x French'
  475 = 'Spare' | German: 'S3 475 Row 48 Spare Message German' | French: 'S3 475 Row 48 Spare Message French'
  476 = 'Spare' | German: 'S3 476 Row 48 Spare Message German' | French: 'S3 476 Row 48 Spare Message French'
  477 = 'Spare' | German: 'S3 477 Row 48 Spare Message German' | French: 'S3 477 Row 48 Spare Message French'
  478 = 'Spare' | German: 'S3 478 Row 48 Spare Message German' | French: 'S3 478 Row 48 Spare Message French'
  479 = 'Spare' | German: 'S3 479 Row 48 Spare Message German' | French: 'S3 479 Row 48 Spare Message French'
  480 = 'Clamp Cylinder A1 Failed to Advance... Check Q1.0...' | German: 'S3 480 Row 49 Failed To Advance.. Check Qxxx.x German' | French: 'S3 480 Row 49 Failed To Advance.. Check Qxxx.x French'
  481 = 'Clamp Cylinder A1 Failed to Return... Check Q1.1...' | German: 'S3 481 Row 49 Failed To Return.. Check Qxxx.x German' | French: 'S3 481 Row 49 Failed To Return.. Check Qxxx.x French'
  482 = 'Clamp Cylinder A1 Lost Advanced... Check I1.0...' | German: 'S3 482 Row 49 Lost Advance Position... Check Ixxx.x German' | French: 'S3 482 Row 49 Lost Advance Position... Check Ixxx.x French'
  483 = 'Clamp Cylinder A1 Lost Returned... Check I1.1...' | German: 'S3 483 Row 49 Lost Return Position... Check Ixxx.x German' | French: 'S3 483 Row 49 Lost Return Position... Check Ixxx.x French'
  484 = 'Clamp Cylinder A1 Switch Fault... Check I1.0, I1.1...' | German: 'S3 484 Row 49 Switch Fault... Check Ixxx.x / Ixxx.x German' | French: 'S3 484 Row 49 Switch Fault... Check Ixxx.x / Ixxx.x French'
  485 = 'Spare' | German: 'S3 485 Row 49 Spare Message German' | French: 'S3 485 Row 49 Spare Message French'
  486 = 'Spare' | German: 'S3 486 Row 49 Spare Message German' | French: 'S3 486 Row 49 Spare Message French'
  487 = 'Spare' | German: 'S3 487 Row 49 Spare Message German' | French: 'S3 487 Row 49 Spare Message French'
  488 = 'Spare' | German: 'S3 488 Row 49 Spare Message German' | French: 'S3 488 Row 49 Spare Message French'
  489 = 'Spare' | German: 'S3 489 Row 49 Spare Message German' | French: 'S3 489 Row 49 Spare Message French'
  490 = 'Clamp Cylinder A1 Failed to Advance... Check Q1.0...' | German: 'S3 490 Row 50 Failed To Advance.. Check Qxxx.x German' | French: 'S3 490 Row 50 Failed To Advance.. Check Qxxx.x French'
  491 = 'Clamp Cylinder A1 Failed to Return... Check Q1.1...' | German: 'S3 491 Row 50 Failed To Return.. Check Qxxx.x German' | French: 'S3 491 Row 50 Failed To Return.. Check Qxxx.x French'
  492 = 'Clamp Cylinder A1 Lost Advanced... Check I1.0...' | German: 'S3 492 Row 50 Lost Advance Position... Check Ixxx.x German' | French: 'S3 492 Row 50 Lost Advance Position... Check Ixxx.x French'
  493 = 'Clamp Cylinder A1 Lost Returned... Check I1.1...' | German: 'S3 493 Row 50 Lost Return Position... Check Ixxx.x German' | French: 'S3 493 Row 50 Lost Return Position... Check Ixxx.x French'
  494 = 'Clamp Cylinder A1 Switch Fault... Check I1.0, I1.1...' | German: 'S3 494 Row 50 Switch Fault... Check Ixxx.x / Ixxx.x German' | French: 'S3 494 Row 50 Switch Fault... Check Ixxx.x / Ixxx.x French'
  495 = 'Spare' | German: 'S3 495 Row 50 Spare Message German' | French: 'S3 495 Row 50 Spare Message French'
  496 = 'Spare' | German: 'S3 496 Row 50 Spare Message German' | French: 'S3 496 Row 50 Spare Message French'
  497 = 'Spare' | German: 'S3 497 Row 50 Spare Message German' | French: 'S3 497 Row 50 Spare Message French'
  498 = 'Spare' | German: 'S3 498 Row 50 Spare Message German' | French: 'S3 498 Row 50 Spare Message French'
  499 = 'Spare' | German: 'S3 499 Row 50 Spare Message German' | French: 'S3 499 Row 50 Spare Message French'
  500 = 'Clamp Cylinder A1 Failed to Advance... Check Q1.0...' | German: 'S3 500 Row 51 Failed To Advance.. Check Qxxx.x German' | French: 'S3 500 Row 51 Failed To Advance.. Check Qxxx.x French'
  501 = 'Clamp Cylinder A1 Failed to Return... Check Q1.1...' | German: 'S3 501 Row 51 Failed To Return.. Check Qxxx.x German' | French: 'S3 501 Row 51 Failed To Return.. Check Qxxx.x French'
  502 = 'Clamp Cylinder A1 Lost Advanced... Check I1.0...' | German: 'S3 502 Row 51 Lost Advance Position... Check Ixxx.x German' | French: 'S3 502 Row 51 Lost Advance Position... Check Ixxx.x French'
  503 = 'Clamp Cylinder A1 Lost Returned... Check I1.1...' | German: 'S3 503 Row 51 Lost Return Position... Check Ixxx.x German' | French: 'S3 503 Row 51 Lost Return Position... Check Ixxx.x French'
  504 = 'Clamp Cylinder A1 Switch Fault... Check I1.0, I1.1...' | German: 'S3 504 Row 51 Switch Fault... Check Ixxx.x / Ixxx.x German' | French: 'S3 504 Row 51 Switch Fault... Check Ixxx.x / Ixxx.x French'
  505 = 'Spare' | German: 'S3 505 Row 51 Spare Message German' | French: 'S3 505 Row 51 Spare Message French'
  506 = 'Spare' | German: 'S3 506 Row 51 Spare Message German' | French: 'S3 506 Row 51 Spare Message French'
  507 = 'Spare' | German: 'S3 507 Row 51 Spare Message German' | French: 'S3 507 Row 51 Spare Message French'
  508 = 'Spare' | German: 'S3 508 Row 51 Spare Message German' | French: 'S3 508 Row 51 Spare Message French'
  509 = 'Spare' | German: 'S3 509 Row 51 Spare Message German' | French: 'S3 509 Row 51 Spare Message French'
  510 = 'Clamp Cylinder A1 Failed to Advance... Check Q1.0...' | German: 'S3 510 Row 52 Failed To Advance.. Check Qxxx.x German' | French: 'S3 510 Row 52 Failed To Advance.. Check Qxxx.x French'
  511 = 'Clamp Cylinder A1 Failed to Return... Check Q1.1...' | German: 'S3 511 Row 52 Failed To Return.. Check Qxxx.x German' | French: 'S3 511 Row 52 Failed To Return.. Check Qxxx.x French'
  512 = 'Clamp Cylinder A1 Lost Advanced... Check I1.0...' | German: 'S3 512 Row 52 Lost Advance Position... Check Ixxx.x German' | French: 'S3 512 Row 52 Lost Advance Position... Check Ixxx.x French'
  513 = 'Clamp Cylinder A1 Lost Returned... Check I1.1...' | German: 'S3 513 Row 52 Lost Return Position... Check Ixxx.x German' | French: 'S3 513 Row 52 Lost Return Position... Check Ixxx.x French'
  514 = 'Clamp Cylinder A1 Switch Fault... Check I1.0, I1.1...' | German: 'S3 514 Row 52 Switch Fault... Check Ixxx.x / Ixxx.x German' | French: 'S3 514 Row 52 Switch Fault... Check Ixxx.x / Ixxx.x French'
  515 = 'Spare' | German: 'S3 515 Row 52 Spare Message German' | French: 'S3 515 Row 52 Spare Message French'
  516 = 'Spare' | German: 'S3 516 Row 52 Spare Message German' | French: 'S3 516 Row 52 Spare Message French'
  517 = 'Spare' | German: 'S3 517 Row 52 Spare Message German' | French: 'S3 517 Row 52 Spare Message French'
  518 = 'Spare' | German: 'S3 518 Row 52 Spare Message German' | French: 'S3 518 Row 52 Spare Message French'
  519 = 'Spare' | German: 'S3 519 Row 52 Spare Message German' | French: 'S3 519 Row 52 Spare Message French'
  520 = 'Clamp Cylinder A1 Failed to Advance... Check Q1.0...' | German: 'S3 520 Row 53 Failed To Advance.. Check Qxxx.x German' | French: 'S3 520 Row 53 Failed To Advance.. Check Qxxx.x French'
  521 = 'Clamp Cylinder A1 Failed to Return... Check Q1.1...' | German: 'S3 521 Row 53 Failed To Return.. Check Qxxx.x German' | French: 'S3 521 Row 53 Failed To Return.. Check Qxxx.x French'
  522 = 'Clamp Cylinder A1 Lost Advanced... Check I1.0...' | German: 'S3 522 Row 53 Lost Advance Position... Check Ixxx.x German' | French: 'S3 522 Row 53 Lost Advance Position... Check Ixxx.x French'
  523 = 'Clamp Cylinder A1 Lost Returned... Check I1.1...' | German: 'S3 523 Row 53 Lost Return Position... Check Ixxx.x German' | French: 'S3 523 Row 53 Lost Return Position... Check Ixxx.x French'
  524 = 'Clamp Cylinder A1 Switch Fault... Check I1.0, I1.1...' | German: 'S3 524 Row 53 Switch Fault... Check Ixxx.x / Ixxx.x German' | French: 'S3 524 Row 53 Switch Fault... Check Ixxx.x / Ixxx.x French'
  525 = 'Spare' | German: 'S3 525 Row 53 Spare Message German' | French: 'S3 525 Row 53 Spare Message French'
  526 = 'Spare' | German: 'S3 526 Row 53 Spare Message German' | French: 'S3 526 Row 53 Spare Message French'
  527 = 'Spare' | German: 'S3 527 Row 53 Spare Message German' | French: 'S3 527 Row 53 Spare Message French'
  528 = 'Spare' | German: 'S3 528 Row 53 Spare Message German' | French: 'S3 528 Row 53 Spare Message French'
  529 = 'Spare' | German: 'S3 529 Row 53 Spare Message German' | French: 'S3 529 Row 53 Spare Message French'
  530 = 'Clamp Cylinder A1 Failed to Advance... Check Q1.0...' | German: 'S3 530 Row 54 Failed To Advance.. Check Qxxx.x German' | French: 'S3 530 Row 54 Failed To Advance.. Check Qxxx.x French'
  531 = 'Clamp Cylinder A1 Failed to Return... Check Q1.1...' | German: 'S3 531 Row 54 Failed To Return.. Check Qxxx.x German' | French: 'S3 531 Row 54 Failed To Return.. Check Qxxx.x French'
  532 = 'Clamp Cylinder A1 Lost Advanced... Check I1.0...' | German: 'S3 532 Row 54 Lost Advance Position... Check Ixxx.x German' | French: 'S3 532 Row 54 Lost Advance Position... Check Ixxx.x French'
  533 = 'Clamp Cylinder A1 Lost Returned... Check I1.1...' | German: 'S3 533 Row 54 Lost Return Position... Check Ixxx.x German' | French: 'S3 533 Row 54 Lost Return Position... Check Ixxx.x French'
  534 = 'Clamp Cylinder A1 Switch Fault... Check I1.0, I1.1...' | German: 'S3 534 Row 54 Switch Fault... Check Ixxx.x / Ixxx.x German' | French: 'S3 534 Row 54 Switch Fault... Check Ixxx.x / Ixxx.x French'
  535 = 'Spare' | German: 'S3 535 Row 54 Spare Message German' | French: 'S3 535 Row 54 Spare Message French'
  536 = 'Spare' | German: 'S3 536 Row 54 Spare Message German' | French: 'S3 536 Row 54 Spare Message French'
  537 = 'Spare' | German: 'S3 537 Row 54 Spare Message German' | French: 'S3 537 Row 54 Spare Message French'
  538 = 'Spare' | German: 'S3 538 Row 54 Spare Message German' | French: 'S3 538 Row 54 Spare Message French'
  539 = 'Spare' | German: 'S3 539 Row 54 Spare Message German' | French: 'S3 539 Row 54 Spare Message French'
  540 = 'Clamp Cylinder A1 Failed to Advance... Check Q1.0...' | German: 'S3 540 Row 55 Failed To Advance.. Check Qxxx.x German' | French: 'S3 540 Row 55 Failed To Advance.. Check Qxxx.x French'
  541 = 'Clamp Cylinder A1 Failed to Return... Check Q1.1...' | German: 'S3 541 Row 55 Failed To Return.. Check Qxxx.x German' | French: 'S3 541 Row 55 Failed To Return.. Check Qxxx.x French'
  542 = 'Clamp Cylinder A1 Lost Advanced... Check I1.0...' | German: 'S3 542 Row 55 Lost Advance Position... Check Ixxx.x German' | French: 'S3 542 Row 55 Lost Advance Position... Check Ixxx.x French'
  543 = 'Clamp Cylinder A1 Lost Returned... Check I1.1...' | German: 'S3 543 Row 55 Lost Return Position... Check Ixxx.x German' | French: 'S3 543 Row 55 Lost Return Position... Check Ixxx.x French'
  544 = 'Clamp Cylinder A1 Switch Fault... Check I1.0, I1.1...' | German: 'S3 544 Row 55 Switch Fault... Check Ixxx.x / Ixxx.x German' | French: 'S3 544 Row 55 Switch Fault... Check Ixxx.x / Ixxx.x French'
  545 = 'Spare' | German: 'S3 545 Row 55 Spare Message German' | French: 'S3 545 Row 55 Spare Message French'
  546 = 'Spare' | German: 'S3 546 Row 55 Spare Message German' | French: 'S3 546 Row 55 Spare Message French'
  547 = 'Spare' | German: 'S3 547 Row 55 Spare Message German' | French: 'S3 547 Row 55 Spare Message French'
  548 = 'Spare' | German: 'S3 548 Row 55 Spare Message German' | French: 'S3 548 Row 55 Spare Message French'
  549 = 'Spare' | German: 'S3 549 Row 55 Spare Message German' | French: 'S3 549 Row 55 Spare Message French'
  550 = 'Clamp Cylinder A1 Failed to Advance... Check Q1.0...' | German: 'S3 550 Row 56 Failed To Advance.. Check Qxxx.x German' | French: 'S3 550 Row 56 Failed To Advance.. Check Qxxx.x French'
  551 = 'Clamp Cylinder A1 Failed to Return... Check Q1.1...' | German: 'S3 551 Row 56 Failed To Return.. Check Qxxx.x German' | French: 'S3 551 Row 56 Failed To Return.. Check Qxxx.x French'
  552 = 'Clamp Cylinder A1 Lost Advanced... Check I1.0...' | German: 'S3 552 Row 56 Lost Advance Position... Check Ixxx.x German' | French: 'S3 552 Row 56 Lost Advance Position... Check Ixxx.x French'
  553 = 'Clamp Cylinder A1 Lost Returned... Check I1.1...' | German: 'S3 553 Row 56 Lost Return Position... Check Ixxx.x German' | French: 'S3 553 Row 56 Lost Return Position... Check Ixxx.x French'
  554 = 'Clamp Cylinder A1 Switch Fault... Check I1.0, I1.1...' | German: 'S3 554 Row 56 Switch Fault... Check Ixxx.x / Ixxx.x German' | French: 'S3 554 Row 56 Switch Fault... Check Ixxx.x / Ixxx.x French'
  555 = 'Spare' | German: 'S3 555 Row 56 Spare Message German' | French: 'S3 555 Row 56 Spare Message French'
  556 = 'Spare' | German: 'S3 556 Row 56 Spare Message German' | French: 'S3 556 Row 56 Spare Message French'
  557 = 'Spare' | German: 'S3 557 Row 56 Spare Message German' | French: 'S3 557 Row 56 Spare Message French'
  558 = 'Spare' | German: 'S3 558 Row 56 Spare Message German' | French: 'S3 558 Row 56 Spare Message French'
  559 = 'Spare' | German: 'S3 559 Row 56 Spare Message German' | French: 'S3 559 Row 56 Spare Message French'
  560 = 'Clamp Cylinder A1 Failed to Advance... Check Q1.0...' | German: 'S3 560 Row 57 Failed To Advance.. Check Qxxx.x German' | French: 'S3 560 Row 57 Failed To Advance.. Check Qxxx.x French'
  561 = 'Clamp Cylinder A1 Failed to Return... Check Q1.1...' | German: 'S3 561 Row 57 Failed To Return.. Check Qxxx.x German' | French: 'S3 561 Row 57 Failed To Return.. Check Qxxx.x French'
  562 = 'Clamp Cylinder A1 Lost Advanced... Check I1.0...' | German: 'S3 562 Row 57 Lost Advance Position... Check Ixxx.x German' | French: 'S3 562 Row 57 Lost Advance Position... Check Ixxx.x French'
  563 = 'Clamp Cylinder A1 Lost Returned... Check I1.1...' | German: 'S3 563 Row 57 Lost Return Position... Check Ixxx.x German' | French: 'S3 563 Row 57 Lost Return Position... Check Ixxx.x French'
  564 = 'Clamp Cylinder A1 Switch Fault... Check I1.0, I1.1...' | German: 'S3 564 Row 57 Switch Fault... Check Ixxx.x / Ixxx.x German' | French: 'S3 564 Row 57 Switch Fault... Check Ixxx.x / Ixxx.x French'
  565 = 'Spare' | German: 'S3 565 Row 57 Spare Message German' | French: 'S3 565 Row 57 Spare Message French'
  566 = 'Spare' | German: 'S3 566 Row 57 Spare Message German' | French: 'S3 566 Row 57 Spare Message French'
  567 = 'Spare' | German: 'S3 567 Row 57 Spare Message German' | French: 'S3 567 Row 57 Spare Message French'
  568 = 'Spare' | German: 'S3 568 Row 57 Spare Message German' | French: 'S3 568 Row 57 Spare Message French'
  569 = 'Spare' | German: 'S3 569 Row 57 Spare Message German' | French: 'S3 569 Row 57 Spare Message French'
  570 = 'Clamp Cylinder A1 Failed to Advance... Check Q1.0...' | German: 'S3 570 Row 58 Failed To Advance.. Check Qxxx.x German' | French: 'S3 570 Row 58 Failed To Advance.. Check Qxxx.x French'
  571 = 'Clamp Cylinder A1 Failed to Return... Check Q1.1...' | German: 'S3 571 Row 58 Failed To Return.. Check Qxxx.x German' | French: 'S3 571 Row 58 Failed To Return.. Check Qxxx.x French'
  572 = 'Clamp Cylinder A1 Lost Advanced... Check I1.0...' | German: 'S3 572 Row 58 Lost Advance Position... Check Ixxx.x German' | French: 'S3 572 Row 58 Lost Advance Position... Check Ixxx.x French'
  573 = 'Clamp Cylinder A1 Lost Returned... Check I1.1...' | German: 'S3 573 Row 58 Lost Return Position... Check Ixxx.x German' | French: 'S3 573 Row 58 Lost Return Position... Check Ixxx.x French'
  574 = 'Clamp Cylinder A1 Switch Fault... Check I1.0, I1.1...' | German: 'S3 574 Row 58 Switch Fault... Check Ixxx.x / Ixxx.x German' | French: 'S3 574 Row 58 Switch Fault... Check Ixxx.x / Ixxx.x French'
  575 = 'Spare' | German: 'S3 575 Row 58 Spare Message German' | French: 'S3 575 Row 58 Spare Message French'
  576 = 'Spare' | German: 'S3 576 Row 58 Spare Message German' | French: 'S3 576 Row 58 Spare Message French'
  577 = 'Spare' | German: 'S3 577 Row 58 Spare Message German' | French: 'S3 577 Row 58 Spare Message French'
  578 = 'Spare' | German: 'S3 578 Row 58 Spare Message German' | French: 'S3 578 Row 58 Spare Message French'
  579 = 'Spare' | German: 'S3 579 Row 58 Spare Message German' | French: 'S3 579 Row 58 Spare Message French'
  580 = 'Clamp Cylinder A1 Failed to Advance... Check Q1.0...' | German: 'S3 580 Row 59 Failed To Advance.. Check Qxxx.x German' | French: 'S3 580 Row 59 Failed To Advance.. Check Qxxx.x French'
  581 = 'Clamp Cylinder A1 Failed to Return... Check Q1.1...' | German: 'S3 581 Row 59 Failed To Return.. Check Qxxx.x German' | French: 'S3 581 Row 59 Failed To Return.. Check Qxxx.x French'
  582 = 'Clamp Cylinder A1 Lost Advanced... Check I1.0...' | German: 'S3 582 Row 59 Lost Advance Position... Check Ixxx.x German' | French: 'S3 582 Row 59 Lost Advance Position... Check Ixxx.x French'
  583 = 'Clamp Cylinder A1 Lost Returned... Check I1.1...' | German: 'S3 583 Row 59 Lost Return Position... Check Ixxx.x German' | French: 'S3 583 Row 59 Lost Return Position... Check Ixxx.x French'
  584 = 'Clamp Cylinder A1 Switch Fault... Check I1.0, I1.1...' | German: 'S3 584 Row 59 Switch Fault... Check Ixxx.x / Ixxx.x German' | French: 'S3 584 Row 59 Switch Fault... Check Ixxx.x / Ixxx.x French'
  585 = 'Spare' | German: 'S3 585 Row 59 Spare Message German' | French: 'S3 585 Row 59 Spare Message French'
  586 = 'Spare' | German: 'S3 586 Row 59 Spare Message German' | French: 'S3 586 Row 59 Spare Message French'
  587 = 'Spare' | German: 'S3 587 Row 59 Spare Message German' | French: 'S3 587 Row 59 Spare Message French'
  588 = 'Spare' | German: 'S3 588 Row 59 Spare Message German' | French: 'S3 588 Row 59 Spare Message French'
  589 = 'Spare' | German: 'S3 589 Row 59 Spare Message German' | French: 'S3 589 Row 59 Spare Message French'
  590 = 'Clamp Cylinder A1 Failed to Advance... Check Q1.0...' | German: 'S3 590 Row 60 Failed To Advance.. Check Qxxx.x German' | French: 'S3 590 Row 60 Failed To Advance.. Check Qxxx.x French'
  591 = 'Clamp Cylinder A1 Failed to Return... Check Q1.1...' | German: 'S3 591 Row 60 Failed To Return.. Check Qxxx.x German' | French: 'S3 591 Row 60 Failed To Return.. Check Qxxx.x French'
  592 = 'Clamp Cylinder A1 Lost Advanced... Check I1.0...' | German: 'S3 592 Row 60 Lost Advance Position... Check Ixxx.x German' | French: 'S3 592 Row 60 Lost Advance Position... Check Ixxx.x French'
  593 = 'Clamp Cylinder A1 Lost Returned... Check I1.1...' | German: 'S3 593 Row 60 Lost Return Position... Check Ixxx.x German' | French: 'S3 593 Row 60 Lost Return Position... Check Ixxx.x French'
  594 = 'Clamp Cylinder A1 Switch Fault... Check I1.0, I1.1...' | German: 'S3 594 Row 60 Switch Fault... Check Ixxx.x / Ixxx.x German' | French: 'S3 594 Row 60 Switch Fault... Check Ixxx.x / Ixxx.x French'
  595 = 'Spare' | German: 'S3 595 Row 60 Spare Message German' | French: 'S3 595 Row 60 Spare Message French'
  596 = 'Spare' | German: 'S3 596 Row 60 Spare Message German' | French: 'S3 596 Row 60 Spare Message French'
  597 = 'Spare' | German: 'S3 597 Row 60 Spare Message German' | French: 'S3 597 Row 60 Spare Message French'
  598 = 'Spare' | German: 'S3 598 Row 60 Spare Message German' | French: 'S3 598 Row 60 Spare Message French'
  599 = 'Spare' | German: 'S3 599 Row 60 Spare Message German' | French: 'S3 599 Row 60 Spare Message French'
  600 = 'Clamp Cylinder A1 Failed to Advance... Check Q1.0...' | German: 'S3 600 Row 61 Failed To Advance.. Check Qxxx.x German' | French: 'S3 600 Row 61 Failed To Advance.. Check Qxxx.x French'
  601 = 'Clamp Cylinder A1 Failed to Return... Check Q1.1...' | German: 'S3 601 Row 61 Failed To Return.. Check Qxxx.x German' | French: 'S3 601 Row 61 Failed To Return.. Check Qxxx.x French'
  602 = 'Clamp Cylinder A1 Lost Advanced... Check I1.0...' | German: 'S3 602 Row 61 Lost Advance Position... Check Ixxx.x German' | French: 'S3 602 Row 61 Lost Advance Position... Check Ixxx.x French'
  603 = 'Clamp Cylinder A1 Lost Returned... Check I1.1...' | German: 'S3 603 Row 61 Lost Return Position... Check Ixxx.x German' | French: 'S3 603 Row 61 Lost Return Position... Check Ixxx.x French'
  604 = 'Clamp Cylinder A1 Switch Fault... Check I1.0, I1.1...' | German: 'S3 604 Row 61 Switch Fault... Check Ixxx.x / Ixxx.x German' | French: 'S3 604 Row 61 Switch Fault... Check Ixxx.x / Ixxx.x French'
  605 = 'Spare' | German: 'S3 605 Row 61 Spare Message German' | French: 'S3 605 Row 61 Spare Message French'
  606 = 'Spare' | German: 'S3 606 Row 61 Spare Message German' | French: 'S3 606 Row 61 Spare Message French'
  607 = 'Spare' | German: 'S3 607 Row 61 Spare Message German' | French: 'S3 607 Row 61 Spare Message French'
  608 = 'Spare' | German: 'S3 608 Row 61 Spare Message German' | French: 'S3 608 Row 61 Spare Message French'
  609 = 'Spare' | German: 'S3 609 Row 61 Spare Message German' | French: 'S3 609 Row 61 Spare Message French'
  610 = 'Clamp Cylinder A1 Failed to Advance... Check Q1.0...' | German: 'S3 610 Row 62 Failed To Advance.. Check Qxxx.x German' | French: 'S3 610 Row 62 Failed To Advance.. Check Qxxx.x French'
  611 = 'Clamp Cylinder A1 Failed to Return... Check Q1.1...' | German: 'S3 611 Row 62 Failed To Return.. Check Qxxx.x German' | French: 'S3 611 Row 62 Failed To Return.. Check Qxxx.x French'
  612 = 'Clamp Cylinder A1 Lost Advanced... Check I1.0...' | German: 'S3 612 Row 62 Lost Advance Position... Check Ixxx.x German' | French: 'S3 612 Row 62 Lost Advance Position... Check Ixxx.x French'
  613 = 'Clamp Cylinder A1 Lost Returned... Check I1.1...' | German: 'S3 613 Row 62 Lost Return Position... Check Ixxx.x German' | French: 'S3 613 Row 62 Lost Return Position... Check Ixxx.x French'
  614 = 'Clamp Cylinder A1 Switch Fault... Check I1.0, I1.1...' | German: 'S3 614 Row 62 Switch Fault... Check Ixxx.x / Ixxx.x German' | French: 'S3 614 Row 62 Switch Fault... Check Ixxx.x / Ixxx.x French'
  615 = 'Spare' | German: 'S3 615 Row 62 Spare Message German' | French: 'S3 615 Row 62 Spare Message French'
  616 = 'Spare' | German: 'S3 616 Row 62 Spare Message German' | French: 'S3 616 Row 62 Spare Message French'
  617 = 'Spare' | German: 'S3 617 Row 62 Spare Message German' | French: 'S3 617 Row 62 Spare Message French'
  618 = 'Spare' | German: 'S3 618 Row 62 Spare Message German' | French: 'S3 618 Row 62 Spare Message French'
  619 = 'Spare' | German: 'S3 619 Row 62 Spare Message German' | French: 'S3 619 Row 62 Spare Message French'
  620 = 'Clamp Cylinder A1 Failed to Advance... Check Q1.0...' | German: 'S3 620 Row 63 Failed To Advance.. Check Qxxx.x German' | French: 'S3 620 Row 63 Failed To Advance.. Check Qxxx.x French'
  621 = 'Clamp Cylinder A1 Failed to Return... Check Q1.1...' | German: 'S3 621 Row 63 Failed To Return.. Check Qxxx.x German' | French: 'S3 621 Row 63 Failed To Return.. Check Qxxx.x French'
  622 = 'Clamp Cylinder A1 Lost Advanced... Check I1.0...' | German: 'S3 622 Row 63 Lost Advance Position... Check Ixxx.x German' | French: 'S3 622 Row 63 Lost Advance Position... Check Ixxx.x French'
  623 = 'Clamp Cylinder A1 Lost Returned... Check I1.1...' | German: 'S3 623 Row 63 Lost Return Position... Check Ixxx.x German' | French: 'S3 623 Row 63 Lost Return Position... Check Ixxx.x French'
  624 = 'Clamp Cylinder A1 Switch Fault... Check I1.0, I1.1...' | German: 'S3 624 Row 63 Switch Fault... Check Ixxx.x / Ixxx.x German' | French: 'S3 624 Row 63 Switch Fault... Check Ixxx.x / Ixxx.x French'
  625 = 'Spare' | German: 'S3 625 Row 63 Spare Message German' | French: 'S3 625 Row 63 Spare Message French'
  626 = 'Spare' | German: 'S3 626 Row 63 Spare Message German' | French: 'S3 626 Row 63 Spare Message French'
  627 = 'Spare' | German: 'S3 627 Row 63 Spare Message German' | French: 'S3 627 Row 63 Spare Message French'
  628 = 'Spare' | German: 'S3 628 Row 63 Spare Message German' | French: 'S3 628 Row 63 Spare Message French'
  629 = 'Spare' | German: 'S3 629 Row 63 Spare Message German' | French: 'S3 629 Row 63 Spare Message French'
  630 = 'Clamp Cylinder A1 Failed to Advance... Check Q1.0...' | German: 'S3 630 Row 64 Failed To Advance.. Check Qxxx.x German' | French: 'S3 630 Row 64 Failed To Advance.. Check Qxxx.x French'
  631 = 'Clamp Cylinder A1 Failed to Return... Check Q1.1...' | German: 'S3 631 Row 64 Failed To Return.. Check Qxxx.x German' | French: 'S3 631 Row 64 Failed To Return.. Check Qxxx.x French'
  632 = 'Clamp Cylinder A1 Lost Advanced... Check I1.0...' | German: 'S3 632 Row 64 Lost Advance Position... Check Ixxx.x German' | French: 'S3 632 Row 64 Lost Advance Position... Check Ixxx.x French'
  633 = 'Clamp Cylinder A1 Lost Returned... Check I1.1...' | German: 'S3 633 Row 64 Lost Return Position... Check Ixxx.x German' | French: 'S3 633 Row 64 Lost Return Position... Check Ixxx.x French'
  634 = 'Clamp Cylinder A1 Switch Fault... Check I1.0, I1.1...' | German: 'S3 634 Row 64 Switch Fault... Check Ixxx.x / Ixxx.x German' | French: 'S3 634 Row 64 Switch Fault... Check Ixxx.x / Ixxx.x French'
  635 = 'Spare' | German: 'S3 635 Row 64 Spare Message German' | French: 'S3 635 Row 64 Spare Message French'
  636 = 'Spare' | German: 'S3 636 Row 64 Spare Message German' | French: 'S3 636 Row 64 Spare Message French'
  637 = 'Spare' | German: 'S3 637 Row 64 Spare Message German' | French: 'S3 637 Row 64 Spare Message French'
  638 = 'Spare' | German: 'S3 638 Row 64 Spare Message German' | French: 'S3 638 Row 64 Spare Message French'
  639 = 'Spare' | German: 'S3 639 Row 64 Spare Message German' | French: 'S3 639 Row 64 Spare Message French'
  640 = 'Clamp Cylinder A1 Failed to Advance... Check Q1.0...' | German: 'S3 640 Row 65 Failed To Advance.. Check Qxxx.x German' | French: 'S3 640 Row 65 Failed To Advance.. Check Qxxx.x French'
  641 = 'Clamp Cylinder A1 Failed to Return... Check Q1.1...' | German: 'S3 641 Row 65 Failed To Return.. Check Qxxx.x German' | French: 'S3 641 Row 65 Failed To Return.. Check Qxxx.x French'
  642 = 'Clamp Cylinder A1 Lost Advanced... Check I1.0...' | German: 'S3 642 Row 65 Lost Advance Position... Check Ixxx.x German' | French: 'S3 642 Row 65 Lost Advance Position... Check Ixxx.x French'
  643 = 'Clamp Cylinder A1 Lost Returned... Check I1.1...' | German: 'S3 643 Row 65 Lost Return Position... Check Ixxx.x German' | French: 'S3 643 Row 65 Lost Return Position... Check Ixxx.x French'
  644 = 'Clamp Cylinder A1 Switch Fault... Check I1.0, I1.1...' | German: 'S3 644 Row 65 Switch Fault... Check Ixxx.x / Ixxx.x German' | French: 'S3 644 Row 65 Switch Fault... Check Ixxx.x / Ixxx.x French'
  645 = 'Spare' | German: 'S3 645 Row 65 Spare Message German' | French: 'S3 645 Row 65 Spare Message French'
  646 = 'Spare' | German: 'S3 646 Row 65 Spare Message German' | French: 'S3 646 Row 65 Spare Message French'
  647 = 'Spare' | German: 'S3 647 Row 65 Spare Message German' | French: 'S3 647 Row 65 Spare Message French'
  648 = 'Spare' | German: 'S3 648 Row 65 Spare Message German' | French: 'S3 648 Row 65 Spare Message French'
  649 = 'Spare' | German: 'S3 649 Row 65 Spare Message German' | French: 'S3 649 Row 65 Spare Message French'
